   1:  PR[GP1:91,1] = PR[GP1:90,1] + -68.704;
   1:  PR[GP1:91,2] = PR[GP1:90,2] + 10.364;
   1:L PR[91] R[100]mm/sec CNT100;
   1:  PR[GP1:91,1] = PR[GP1:90,1] + -68.768;
   1:  PR[GP1:91,2] = PR[GP1:90,2] + 10.145;
   1:L PR[91] R[100]mm/sec CNT100;
   1:  PR[GP1:91,1] = PR[GP1:90,1] + -70.361;
   1:  PR[GP1:91,2] = PR[GP1:90,2] + -0.071;
   1:L PR[91] R[100]mm/sec CNT100;
   1:  PR[GP1:91,1] = PR[GP1:90,1] + -68.787;
   1:  PR[GP1:91,2] = PR[GP1:90,2] + -10.040;
   1:L PR[91] R[100]mm/sec CNT100;
   1:  PR[GP1:91,1] = PR[GP1:90,1] + -68.763;
   1:  PR[GP1:91,2] = PR[GP1:90,2] + -10.308;
   1:L PR[91] R[100]mm/sec CNT100;
   1:  PR[GP1:91,1] = PR[GP1:90,1] + -68.704;
   1:  PR[GP1:91,2] = PR[GP1:90,2] + -10.508;
   1:L PR[91] R[100]mm/sec CNT100;
   1:  PR[GP1:91,1] = PR[GP1:90,1] + -64.096;
   1:  PR[GP1:91,2] = PR[GP1:90,2] + -19.722;
   1:L PR[91] R[100]mm/sec CNT100;
   1:  PR[GP1:91,1] = PR[GP1:90,1] + -63.563;
   1:  PR[GP1:91,2] = PR[GP1:90,2] + -20.414;
   1:L PR[91] R[100]mm/sec CNT100;
   1:  PR[GP1:91,1] = PR[GP1:90,1] + -57.623;
   1:  PR[GP1:91,2] = PR[GP1:90,2] + -26.659;
   1:L PR[91] R[100]mm/sec CNT100;
   1:  PR[GP1:91,1] = PR[GP1:90,1] + -56.395;
   1:  PR[GP1:91,2] = PR[GP1:90,2] + -27.760;
   1:L PR[91] R[100]mm/sec CNT100;
   1:  PR[GP1:91,1] = PR[GP1:90,1] + -50.541;
   1:  PR[GP1:91,2] = PR[GP1:90,2] + -31.053;
   1:L PR[91] R[100]mm/sec CNT100;
   1:  PR[GP1:91,1] = PR[GP1:90,1] + -48.442;
   1:  PR[GP1:91,2] = PR[GP1:90,2] + -32.383;
   1:L PR[91] R[100]mm/sec CNT100;
   1:  PR[GP1:91,1] = PR[GP1:90,1] + -45.404;
   1:  PR[GP1:91,2] = PR[GP1:90,2] + -33.579;
   1:L PR[91] R[100]mm/sec CNT100;
   1:  PR[GP1:91,1] = PR[GP1:90,1] + -41.020;
   1:  PR[GP1:91,2] = PR[GP1:90,2] + -34.610;
   1:L PR[91] R[100]mm/sec CNT100;
   1:  PR[GP1:91,1] = PR[GP1:90,1] + -37.021;
   1:  PR[GP1:91,2] = PR[GP1:90,2] + -35.453;
   1:L PR[91] R[100]mm/sec CNT100;
   1:  PR[GP1:91,1] = PR[GP1:90,1] + -31.107;
   1:  PR[GP1:91,2] = PR[GP1:90,2] + -35.621;
   1:L PR[91] R[100]mm/sec CNT100;
   1:  PR[GP1:91,1] = PR[GP1:90,1] + -30.091;
   1:  PR[GP1:91,2] = PR[GP1:90,2] + -35.570;
   1:L PR[91] R[100]mm/sec CNT100;
   1:  PR[GP1:91,1] = PR[GP1:90,1] + -27.280;
   1:  PR[GP1:91,2] = PR[GP1:90,2] + -35.161;
   1:L PR[91] R[100]mm/sec CNT100;
   1:  PR[GP1:91,1] = PR[GP1:90,1] + -23.789;
   1:  PR[GP1:91,2] = PR[GP1:90,2] + -34.705;
   1:L PR[91] R[100]mm/sec CNT100;
   1:  PR[GP1:91,1] = PR[GP1:90,1] + -17.856;
   1:  PR[GP1:91,2] = PR[GP1:90,2] + -32.817;
   1:L PR[91] R[100]mm/sec CNT100;
   1:  PR[GP1:91,1] = PR[GP1:90,1] + -16.773;
   1:  PR[GP1:91,2] = PR[GP1:90,2] + -32.440;
   1:L PR[91] R[100]mm/sec CNT100;
   1:  PR[GP1:91,1] = PR[GP1:90,1] + -11.344;
   1:  PR[GP1:91,2] = PR[GP1:90,2] + -29.600;
   1:L PR[91] R[100]mm/sec CNT100;
   1:  PR[GP1:91,1] = PR[GP1:90,1] + -10.310;
   1:  PR[GP1:91,2] = PR[GP1:90,2] + -28.848;
   1:L PR[91] R[100]mm/sec CNT100;
   1:  PR[GP1:91,1] = PR[GP1:90,1] + -6.534;
   1:  PR[GP1:91,2] = PR[GP1:90,2] + -25.891;
   1:L PR[91] R[100]mm/sec CNT100;
   1:  PR[GP1:91,1] = PR[GP1:90,1] + -3.696;
   1:  PR[GP1:91,2] = PR[GP1:90,2] + -22.600;
   1:L PR[91] R[100]mm/sec CNT100;
   1:  PR[GP1:91,1] = PR[GP1:90,1] + -2.135;
   1:  PR[GP1:91,2] = PR[GP1:90,2] + -22.265;
   1:L PR[91] R[100]mm/sec CNT100;
   1:  PR[GP1:91,1] = PR[GP1:90,1] + 0.475;
   1:  PR[GP1:91,2] = PR[GP1:90,2] + -20.882;
   1:L PR[91] R[100]mm/sec CNT100;
   1:  PR[GP1:91,1] = PR[GP1:90,1] + 3.972;
   1:  PR[GP1:91,2] = PR[GP1:90,2] + -22.663;
   1:L PR[91] R[100]mm/sec CNT100;
   1:  PR[GP1:91,1] = PR[GP1:90,1] + 6.781;
   1:  PR[GP1:91,2] = PR[GP1:90,2] + -25.925;
   1:L PR[91] R[100]mm/sec CNT100;
   1:  PR[GP1:91,1] = PR[GP1:90,1] + 10.539;
   1:  PR[GP1:91,2] = PR[GP1:90,2] + -28.865;
   1:L PR[91] R[100]mm/sec CNT100;
   1:  PR[GP1:91,1] = PR[GP1:90,1] + 11.575;
   1:  PR[GP1:91,2] = PR[GP1:90,2] + -29.617;
   1:L PR[91] R[100]mm/sec CNT100;
   1:  PR[GP1:91,1] = PR[GP1:90,1] + 16.965;
   1:  PR[GP1:91,2] = PR[GP1:90,2] + -32.430;
   1:L PR[91] R[100]mm/sec CNT100;
   1:  PR[GP1:91,1] = PR[GP1:90,1] + 23.998;
   1:  PR[GP1:91,2] = PR[GP1:90,2] + -34.701;
   1:L PR[91] R[100]mm/sec CNT100;
   1:  PR[GP1:91,1] = PR[GP1:90,1] + 27.494;
   1:  PR[GP1:91,2] = PR[GP1:90,2] + -35.160;
   1:L PR[91] R[100]mm/sec CNT100;
   1:  PR[GP1:91,1] = PR[GP1:90,1] + 30.293;
   1:  PR[GP1:91,2] = PR[GP1:90,2] + -35.570;
   1:L PR[91] R[100]mm/sec CNT100;
   1:  PR[GP1:91,1] = PR[GP1:90,1] + 31.306;
   1:  PR[GP1:91,2] = PR[GP1:90,2] + -35.621;
   1:L PR[91] R[100]mm/sec CNT100;
   1:  PR[GP1:91,1] = PR[GP1:90,1] + 37.198;
   1:  PR[GP1:91,2] = PR[GP1:90,2] + -35.458;
   1:L PR[91] R[100]mm/sec CNT100;
   1:  PR[GP1:91,1] = PR[GP1:90,1] + 40.845;
   1:  PR[GP1:91,2] = PR[GP1:90,2] + -34.609;
   1:L PR[91] R[100]mm/sec CNT100;
   1:  PR[GP1:91,1] = PR[GP1:90,1] + 45.595;
   1:  PR[GP1:91,2] = PR[GP1:90,2] + -33.581;
   1:L PR[91] R[100]mm/sec CNT100;
   1:  PR[GP1:91,1] = PR[GP1:90,1] + 48.654;
   1:  PR[GP1:91,2] = PR[GP1:90,2] + -32.384;
   1:L PR[91] R[100]mm/sec CNT100;
   1:  PR[GP1:91,1] = PR[GP1:90,1] + 54.661;
   1:  PR[GP1:91,2] = PR[GP1:90,2] + -28.971;
   1:L PR[91] R[100]mm/sec CNT100;
   1:  PR[GP1:91,1] = PR[GP1:90,1] + 56.580;
   1:  PR[GP1:91,2] = PR[GP1:90,2] + -27.789;
   1:L PR[91] R[100]mm/sec CNT100;
   1:  PR[GP1:91,1] = PR[GP1:90,1] + 57.816;
   1:  PR[GP1:91,2] = PR[GP1:90,2] + -26.683;
   1:L PR[91] R[100]mm/sec CNT100;
   1:  PR[GP1:91,1] = PR[GP1:90,1] + 63.762;
   1:  PR[GP1:91,2] = PR[GP1:90,2] + -20.413;
   1:L PR[91] R[100]mm/sec CNT100;
   1:  PR[GP1:91,1] = PR[GP1:90,1] + 64.305;
   1:  PR[GP1:91,2] = PR[GP1:90,2] + -19.711;
   1:L PR[91] R[100]mm/sec CNT100;
   1:  PR[GP1:91,1] = PR[GP1:90,1] + 68.916;
   1:  PR[GP1:91,2] = PR[GP1:90,2] + -10.539;
   1:L PR[91] R[100]mm/sec CNT100;
   1:  PR[GP1:91,1] = PR[GP1:90,1] + 68.980;
   1:  PR[GP1:91,2] = PR[GP1:90,2] + -10.324;
   1:L PR[91] R[100]mm/sec CNT100;
   1:  PR[GP1:91,1] = PR[GP1:90,1] + 70.574;
   1:  PR[GP1:91,2] = PR[GP1:90,2] + -0.073;
   1:L PR[91] R[100]mm/sec CNT100;
   1:  PR[GP1:91,1] = PR[GP1:90,1] + 69.000;
   1:  PR[GP1:91,2] = PR[GP1:90,2] + 9.923;
   1:L PR[91] R[100]mm/sec CNT100;
   1:  PR[GP1:91,1] = PR[GP1:90,1] + 68.975;
   1:  PR[GP1:91,2] = PR[GP1:90,2] + 10.199;
   1:L PR[91] R[100]mm/sec CNT100;
   1:  PR[GP1:91,1] = PR[GP1:90,1] + 68.916;
   1:  PR[GP1:91,2] = PR[GP1:90,2] + 10.395;
   1:L PR[91] R[100]mm/sec CNT100;
   1:  PR[GP1:91,1] = PR[GP1:90,1] + 64.305;
   1:  PR[GP1:91,2] = PR[GP1:90,2] + 19.567;
   1:L PR[91] R[100]mm/sec CNT100;
   1:  PR[GP1:91,1] = PR[GP1:90,1] + 63.762;
   1:  PR[GP1:91,2] = PR[GP1:90,2] + 20.269;
   1:L PR[91] R[100]mm/sec CNT100;
   1:  PR[GP1:91,1] = PR[GP1:90,1] + 57.816;
   1:  PR[GP1:91,2] = PR[GP1:90,2] + 26.539;
   1:L PR[91] R[100]mm/sec CNT100;
   1:  PR[GP1:91,1] = PR[GP1:90,1] + 56.589;
   1:  PR[GP1:91,2] = PR[GP1:90,2] + 27.636;
   1:L PR[91] R[100]mm/sec CNT100;
   1:  PR[GP1:91,1] = PR[GP1:90,1] + 50.734;
   1:  PR[GP1:91,2] = PR[GP1:90,2] + 30.926;
   1:L PR[91] R[100]mm/sec CNT100;
   1:  PR[GP1:91,1] = PR[GP1:90,1] + 48.641;
   1:  PR[GP1:91,2] = PR[GP1:90,2] + 32.245;
   1:L PR[91] R[100]mm/sec CNT100;
   1:  PR[GP1:91,1] = PR[GP1:90,1] + 45.590;
   1:  PR[GP1:91,2] = PR[GP1:90,2] + 33.439;
   1:L PR[91] R[100]mm/sec CNT100;
   1:  PR[GP1:91,1] = PR[GP1:90,1] + 41.209;
   1:  PR[GP1:91,2] = PR[GP1:90,2] + 34.472;
   1:L PR[91] R[100]mm/sec CNT100;
   1:  PR[GP1:91,1] = PR[GP1:90,1] + 37.204;
   1:  PR[GP1:91,2] = PR[GP1:90,2] + 35.314;
   1:L PR[91] R[100]mm/sec CNT100;
   1:  PR[GP1:91,1] = PR[GP1:90,1] + 31.306;
   1:  PR[GP1:91,2] = PR[GP1:90,2] + 35.477;
   1:L PR[91] R[100]mm/sec CNT100;
   1:  PR[GP1:91,1] = PR[GP1:90,1] + 30.293;
   1:  PR[GP1:91,2] = PR[GP1:90,2] + 35.426;
   1:L PR[91] R[100]mm/sec CNT100;
   1:  PR[GP1:91,1] = PR[GP1:90,1] + 27.494;
   1:  PR[GP1:91,2] = PR[GP1:90,2] + 35.016;
   1:L PR[91] R[100]mm/sec CNT100;
   1:  PR[GP1:91,1] = PR[GP1:90,1] + 23.998;
   1:  PR[GP1:91,2] = PR[GP1:90,2] + 34.557;
   1:L PR[91] R[100]mm/sec CNT100;
   1:  PR[GP1:91,1] = PR[GP1:90,1] + 18.058;
   1:  PR[GP1:91,2] = PR[GP1:90,2] + 32.667;
   1:L PR[91] R[100]mm/sec CNT100;
   1:  PR[GP1:91,1] = PR[GP1:90,1] + 16.973;
   1:  PR[GP1:91,2] = PR[GP1:90,2] + 32.291;
   1:L PR[91] R[100]mm/sec CNT100;
   1:  PR[GP1:91,1] = PR[GP1:90,1] + 11.573;
   1:  PR[GP1:91,2] = PR[GP1:90,2] + 29.473;
   1:L PR[91] R[100]mm/sec CNT100;
   1:  PR[GP1:91,1] = PR[GP1:90,1] + 10.831;
   1:  PR[GP1:91,2] = PR[GP1:90,2] + 28.949;
   1:L PR[91] R[100]mm/sec CNT100;
   1:  PR[GP1:91,1] = PR[GP1:90,1] + 6.935;
   1:  PR[GP1:91,2] = PR[GP1:90,2] + 25.900;
   1:L PR[91] R[100]mm/sec CNT100;
   1:  PR[GP1:91,1] = PR[GP1:90,1] + 3.954;
   1:  PR[GP1:91,2] = PR[GP1:90,2] + 22.430;
   1:L PR[91] R[100]mm/sec CNT100;
   1:  PR[GP1:91,1] = PR[GP1:90,1] + 3.223;
   1:  PR[GP1:91,2] = PR[GP1:90,2] + 22.142;
   1:L PR[91] R[100]mm/sec CNT100;
   1:  PR[GP1:91,1] = PR[GP1:90,1] + 0.588;
   1:  PR[GP1:91,2] = PR[GP1:90,2] + 20.795;
   1:L PR[91] R[100]mm/sec CNT100;
   1:  ! -- Layer/Ebene 72 -- !;
   1:  PR[91] = PR[90];
   1:  PR[GP1:91,1] = PR[GP1:90,1] + -0.946;
   1:  PR[GP1:91,2] = PR[GP1:90,2] + 21.328;
   1:  PR[GP1:91,3] = PR[GP1:90,3] + 44.225;
   1:L PR[91] R[100]mm/sec CNT100;
   1:  PR[GP1:91,1] = PR[GP1:90,1] + -3.723;
   1:  PR[GP1:91,2] = PR[GP1:90,2] + 22.740;
   1:L PR[91] R[100]mm/sec CNT100;
   1:  PR[GP1:91,1] = PR[GP1:90,1] + -6.531;
   1:  PR[GP1:91,2] = PR[GP1:90,2] + 26.005;
   1:L PR[91] R[100]mm/sec CNT100;
   1:  PR[GP1:91,1] = PR[GP1:90,1] + -10.272;
   1:  PR[GP1:91,2] = PR[GP1:90,2] + 28.935;
   1:L PR[91] R[100]mm/sec CNT100;
   1:  PR[GP1:91,1] = PR[GP1:90,1] + -11.131;
   1:  PR[GP1:91,2] = PR[GP1:90,2] + 29.542;
   1:L PR[91] R[100]mm/sec CNT100;
   1:  PR[GP1:91,1] = PR[GP1:90,1] + -16.427;
   1:  PR[GP1:91,2] = PR[GP1:90,2] + 32.313;
   1:L PR[91] R[100]mm/sec CNT100;
   1:  PR[GP1:91,1] = PR[GP1:90,1] + -22.908;
   1:  PR[GP1:91,2] = PR[GP1:90,2] + 34.395;
   1:L PR[91] R[100]mm/sec CNT100;
   1:  PR[GP1:91,1] = PR[GP1:90,1] + -23.599;
   1:  PR[GP1:91,2] = PR[GP1:90,2] + 34.634;
   1:L PR[91] R[100]mm/sec CNT100;
   1:  PR[GP1:91,1] = PR[GP1:90,1] + -30.227;
   1:  PR[GP1:91,2] = PR[GP1:90,2] + 35.511;
   1:L PR[91] R[100]mm/sec CNT100;
   1:  PR[GP1:91,1] = PR[GP1:90,1] + -30.457;
   1:  PR[GP1:91,2] = PR[GP1:90,2] + 35.523;
   1:L PR[91] R[100]mm/sec CNT100;
   1:  PR[GP1:91,1] = PR[GP1:90,1] + -36.896;
   1:  PR[GP1:91,2] = PR[GP1:90,2] + 35.340;
   1:L PR[91] R[100]mm/sec CNT100;
   1:  PR[GP1:91,1] = PR[GP1:90,1] + -39.667;
   1:  PR[GP1:91,2] = PR[GP1:90,2] + 34.695;
   1:L PR[91] R[100]mm/sec CNT100;
   1:  PR[GP1:91,1] = PR[GP1:90,1] + -45.015;
   1:  PR[GP1:91,2] = PR[GP1:90,2] + 33.536;
   1:L PR[91] R[100]mm/sec CNT100;
   1:  PR[GP1:91,1] = PR[GP1:90,1] + -48.459;
   1:  PR[GP1:91,2] = PR[GP1:90,2] + 32.181;
   1:L PR[91] R[100]mm/sec CNT100;
   1:  PR[GP1:91,1] = PR[GP1:90,1] + -53.838;
   1:  PR[GP1:91,2] = PR[GP1:90,2] + 29.120;
   1:L PR[91] R[100]mm/sec CNT100;
   1:  PR[GP1:91,1] = PR[GP1:90,1] + -56.172;
   1:  PR[GP1:91,2] = PR[GP1:90,2] + 27.675;
   1:L PR[91] R[100]mm/sec CNT100;
   1:  PR[GP1:91,1] = PR[GP1:90,1] + -57.679;
   1:  PR[GP1:91,2] = PR[GP1:90,2] + 26.324;
   1:L PR[91] R[100]mm/sec CNT100;
   1:  PR[GP1:91,1] = PR[GP1:90,1] + -63.196;
   1:  PR[GP1:91,2] = PR[GP1:90,2] + 20.524;
   1:L PR[91] R[100]mm/sec CNT100;
   1:  PR[GP1:91,1] = PR[GP1:90,1] + -63.972;
   1:  PR[GP1:91,2] = PR[GP1:90,2] + 19.517;
   1:L PR[91] R[100]mm/sec CNT100;
   1:  PR[GP1:91,1] = PR[GP1:90,1] + -68.487;
   1:  PR[GP1:91,2] = PR[GP1:90,2] + 10.491;
   1:L PR[91] R[100]mm/sec CNT100;
   1:  PR[GP1:91,1] = PR[GP1:90,1] + -68.652;
   1:  PR[GP1:91,2] = PR[GP1:90,2] + 9.931;
   1:L PR[91] R[100]mm/sec CNT100;
   1:  PR[GP1:91,1] = PR[GP1:90,1] + -70.166;
   1:  PR[GP1:91,2] = PR[GP1:90,2] + 0.222;
   1:L PR[91] R[100]mm/sec CNT100;
   1:  PR[GP1:91,1] = PR[GP1:90,1] + -70.190;
   1:  PR[GP1:91,2] = PR[GP1:90,2] + -0.052;
   1:L PR[91] R[100]mm/sec CNT100;
   1:  PR[GP1:91,1] = PR[GP1:90,1] + -68.700;
   1:  PR[GP1:91,2] = PR[GP1:90,2] + -9.487;
   1:L PR[91] R[100]mm/sec CNT100;
   1:  PR[GP1:91,1] = PR[GP1:90,1] + -68.646;
   1:  PR[GP1:91,2] = PR[GP1:90,2] + -10.094;
   1:L PR[91] R[100]mm/sec CNT100;
   1:  PR[GP1:91,1] = PR[GP1:90,1] + -68.487;
   1:  PR[GP1:91,2] = PR[GP1:90,2] + -10.635;
   1:L PR[91] R[100]mm/sec CNT100;
   1:  PR[GP1:91,1] = PR[GP1:90,1] + -63.972;
   1:  PR[GP1:91,2] = PR[GP1:90,2] + -19.661;
   1:L PR[91] R[100]mm/sec CNT100;
   1:  PR[GP1:91,1] = PR[GP1:90,1] + -63.196;
   1:  PR[GP1:91,2] = PR[GP1:90,2] + -20.668;
   1:L PR[91] R[100]mm/sec CNT100;
   1:  PR[GP1:91,1] = PR[GP1:90,1] + -57.679;
   1:  PR[GP1:91,2] = PR[GP1:90,2] + -26.468;
   1:L PR[91] R[100]mm/sec CNT100;
   1:  PR[GP1:91,1] = PR[GP1:90,1] + -56.181;
   1:  PR[GP1:91,2] = PR[GP1:90,2] + -27.810;
   1:L PR[91] R[100]mm/sec CNT100;
   1:  PR[GP1:91,1] = PR[GP1:90,1] + -50.817;
   1:  PR[GP1:91,2] = PR[GP1:90,2] + -30.828;
   1:L PR[91] R[100]mm/sec CNT100;
   1:  PR[GP1:91,1] = PR[GP1:90,1] + -48.446;
   1:  PR[GP1:91,2] = PR[GP1:90,2] + -32.330;
   1:L PR[91] R[100]mm/sec CNT100;
   1:  PR[GP1:91,1] = PR[GP1:90,1] + -45.010;
   1:  PR[GP1:91,2] = PR[GP1:90,2] + -33.682;
   1:L PR[91] R[100]mm/sec CNT100;
   1:  PR[GP1:91,1] = PR[GP1:90,1] + -41.261;
   1:  PR[GP1:91,2] = PR[GP1:90,2] + -34.565;
   1:L PR[91] R[100]mm/sec CNT100;
   1:  PR[GP1:91,1] = PR[GP1:90,1] + -36.902;
   1:  PR[GP1:91,2] = PR[GP1:90,2] + -35.483;
   1:L PR[91] R[100]mm/sec CNT100;
   1:  PR[GP1:91,1] = PR[GP1:90,1] + -30.457;
   1:  PR[GP1:91,2] = PR[GP1:90,2] + -35.667;
   1:L PR[91] R[100]mm/sec CNT100;
   1:  PR[GP1:91,1] = PR[GP1:90,1] + -30.227;
   1:  PR[GP1:91,2] = PR[GP1:90,2] + -35.655;
   1:L PR[91] R[100]mm/sec CNT100;
   1:  PR[GP1:91,1] = PR[GP1:90,1] + -23.591;
   1:  PR[GP1:91,2] = PR[GP1:90,2] + -34.777;
   1:L PR[91] R[100]mm/sec CNT100;
   1:  PR[GP1:91,1] = PR[GP1:90,1] + -17.788;
   1:  PR[GP1:91,2] = PR[GP1:90,2] + -32.930;
   1:L PR[91] R[100]mm/sec CNT100;
   1:  PR[GP1:91,1] = PR[GP1:90,1] + -16.431;
   1:  PR[GP1:91,2] = PR[GP1:90,2] + -32.459;
   1:L PR[91] R[100]mm/sec CNT100;
   1:  PR[GP1:91,1] = PR[GP1:90,1] + -11.133;
   1:  PR[GP1:91,2] = PR[GP1:90,2] + -29.687;
   1:L PR[91] R[100]mm/sec CNT100;
   1:  PR[GP1:91,1] = PR[GP1:90,1] + -9.935;
   1:  PR[GP1:91,2] = PR[GP1:90,2] + -28.817;
   1:L PR[91] R[100]mm/sec CNT100;
   1:  PR[GP1:91,1] = PR[GP1:90,1] + -6.361;
   1:  PR[GP1:91,2] = PR[GP1:90,2] + -26.017;
   1:L PR[91] R[100]mm/sec CNT100;
   1:  PR[GP1:91,1] = PR[GP1:90,1] + -3.667;
   1:  PR[GP1:91,2] = PR[GP1:90,2] + -22.893;
   1:L PR[91] R[100]mm/sec CNT100;
   1:  PR[GP1:91,1] = PR[GP1:90,1] + -1.968;
   1:  PR[GP1:91,2] = PR[GP1:90,2] + -22.529;
   1:L PR[91] R[100]mm/sec CNT100;
   1:  PR[GP1:91,1] = PR[GP1:90,1] + 0.517;
   1:  PR[GP1:91,2] = PR[GP1:90,2] + -21.212;
   1:L PR[91] R[100]mm/sec CNT100;
   1:  PR[GP1:91,1] = PR[GP1:90,1] + 3.942;
   1:  PR[GP1:91,2] = PR[GP1:90,2] + -22.956;
   1:L PR[91] R[100]mm/sec CNT100;
   1:  PR[GP1:91,1] = PR[GP1:90,1] + 6.606;
   1:  PR[GP1:91,2] = PR[GP1:90,2] + -26.049;
   1:L PR[91] R[100]mm/sec CNT100;
   1:  PR[GP1:91,1] = PR[GP1:90,1] + 10.164;
   1:  PR[GP1:91,2] = PR[GP1:90,2] + -28.833;
   1:L PR[91] R[100]mm/sec CNT100;
   1:  PR[GP1:91,1] = PR[GP1:90,1] + 11.363;
   1:  PR[GP1:91,2] = PR[GP1:90,2] + -29.704;
   1:L PR[91] R[100]mm/sec CNT100;
   1:  PR[GP1:91,1] = PR[GP1:90,1] + 16.623;
   1:  PR[GP1:91,2] = PR[GP1:90,2] + -32.449;
   1:L PR[91] R[100]mm/sec CNT100;
   1:  PR[GP1:91,1] = PR[GP1:90,1] + 23.114;
   1:  PR[GP1:91,2] = PR[GP1:90,2] + -34.534;
   1:L PR[91] R[100]mm/sec CNT100;
   1:  PR[GP1:91,1] = PR[GP1:90,1] + 23.806;
   1:  PR[GP1:91,2] = PR[GP1:90,2] + -34.774;
   1:L PR[91] R[100]mm/sec CNT100;
   1:  PR[GP1:91,1] = PR[GP1:90,1] + 30.428;
   1:  PR[GP1:91,2] = PR[GP1:90,2] + -35.655;
   1:L PR[91] R[100]mm/sec CNT100;
   1:  PR[GP1:91,1] = PR[GP1:90,1] + 30.654;
   1:  PR[GP1:91,2] = PR[GP1:90,2] + -35.667;
   1:L PR[91] R[100]mm/sec CNT100;
   1:  PR[GP1:91,1] = PR[GP1:90,1] + 37.075;
   1:  PR[GP1:91,2] = PR[GP1:90,2] + -35.488;
   1:L PR[91] R[100]mm/sec CNT100;
   1:  PR[GP1:91,1] = PR[GP1:90,1] + 39.837;
   1:  PR[GP1:91,2] = PR[GP1:90,2] + -34.846;
   1:L PR[91] R[100]mm/sec CNT100;
   1:  PR[GP1:91,1] = PR[GP1:90,1] + 45.197;
   1:  PR[GP1:91,2] = PR[GP1:90,2] + -33.686;
   1:L PR[91] R[100]mm/sec CNT100;
   1:  PR[GP1:91,1] = PR[GP1:90,1] + 48.657;
   1:  PR[GP1:91,2] = PR[GP1:90,2] + -32.332;
   1:L PR[91] R[100]mm/sec CNT100;
   1:  PR[GP1:91,1] = PR[GP1:90,1] + 54.035;
   1:  PR[GP1:91,2] = PR[GP1:90,2] + -29.277;
   1:L PR[91] R[100]mm/sec CNT100;
   1:  PR[GP1:91,1] = PR[GP1:90,1] + 56.363;
   1:  PR[GP1:91,2] = PR[GP1:90,2] + -27.841;
   1:L PR[91] R[100]mm/sec CNT100;
   1:  PR[GP1:91,1] = PR[GP1:90,1] + 57.868;
   1:  PR[GP1:91,2] = PR[GP1:90,2] + -26.496;
   1:L PR[91] R[100]mm/sec CNT100;
   1:  PR[GP1:91,1] = PR[GP1:90,1] + 63.389;
   1:  PR[GP1:91,2] = PR[GP1:90,2] + -20.673;
   1:L PR[91] R[100]mm/sec CNT100;
   1:  PR[GP1:91,1] = PR[GP1:90,1] + 64.178;
   1:  PR[GP1:91,2] = PR[GP1:90,2] + -19.653;
   1:L PR[91] R[100]mm/sec CNT100;
   1:  PR[GP1:91,1] = PR[GP1:90,1] + 68.698;
   1:  PR[GP1:91,2] = PR[GP1:90,2] + -10.669;
   1:L PR[91] R[100]mm/sec CNT100;
   1:  PR[GP1:91,1] = PR[GP1:90,1] + 68.862;
   1:  PR[GP1:91,2] = PR[GP1:90,2] + -10.118;
   1:L PR[91] R[100]mm/sec CNT100;
   1:  PR[GP1:91,1] = PR[GP1:90,1] + 70.377;
   1:  PR[GP1:91,2] = PR[GP1:90,2] + -0.376;
   1:L PR[91] R[100]mm/sec CNT100;
   1:  PR[GP1:91,1] = PR[GP1:90,1] + 70.403;
   1:  PR[GP1:91,2] = PR[GP1:90,2] + -0.092;
   1:L PR[91] R[100]mm/sec CNT100;
   1:  PR[GP1:91,1] = PR[GP1:90,1] + 68.913;
   1:  PR[GP1:91,2] = PR[GP1:90,2] + 9.368;
   1:L PR[91] R[100]mm/sec CNT100;
   1:  PR[GP1:91,1] = PR[GP1:90,1] + 68.857;
   1:  PR[GP1:91,2] = PR[GP1:90,2] + 9.993;
   1:L PR[91] R[100]mm/sec CNT100;
   1:  PR[GP1:91,1] = PR[GP1:90,1] + 68.698;
   1:  PR[GP1:91,2] = PR[GP1:90,2] + 10.525;
   1:L PR[91] R[100]mm/sec CNT100;
   1:  PR[GP1:91,1] = PR[GP1:90,1] + 64.178;
   1:  PR[GP1:91,2] = PR[GP1:90,2] + 19.509;
   1:L PR[91] R[100]mm/sec CNT100;
   1:  PR[GP1:91,1] = PR[GP1:90,1] + 63.389;
   1:  PR[GP1:91,2] = PR[GP1:90,2] + 20.529;
   1:L PR[91] R[100]mm/sec CNT100;
   1:  PR[GP1:91,1] = PR[GP1:90,1] + 57.868;
   1:  PR[GP1:91,2] = PR[GP1:90,2] + 26.352;
   1:L PR[91] R[100]mm/sec CNT100;
   1:  PR[GP1:91,1] = PR[GP1:90,1] + 56.372;
   1:  PR[GP1:91,2] = PR[GP1:90,2] + 27.689;
   1:L PR[91] R[100]mm/sec CNT100;
   1:  PR[GP1:91,1] = PR[GP1:90,1] + 51.007;
   1:  PR[GP1:91,2] = PR[GP1:90,2] + 30.704;
   1:L PR[91] R[100]mm/sec CNT100;
   1:  PR[GP1:91,1] = PR[GP1:90,1] + 48.644;
   1:  PR[GP1:91,2] = PR[GP1:90,2] + 32.193;
   1:L PR[91] R[100]mm/sec CNT100;
   1:  PR[GP1:91,1] = PR[GP1:90,1] + 45.192;
   1:  PR[GP1:91,2] = PR[GP1:90,2] + 33.544;
   1:L PR[91] R[100]mm/sec CNT100;
   1:  PR[GP1:91,1] = PR[GP1:90,1] + 41.447;
   1:  PR[GP1:91,2] = PR[GP1:90,2] + 34.427;
   1:L PR[91] R[100]mm/sec CNT100;
   1:  PR[GP1:91,1] = PR[GP1:90,1] + 37.082;
   1:  PR[GP1:91,2] = PR[GP1:90,2] + 35.344;
   1:L PR[91] R[100]mm/sec CNT100;
   1:  PR[GP1:91,1] = PR[GP1:90,1] + 30.654;
   1:  PR[GP1:91,2] = PR[GP1:90,2] + 35.523;
   1:L PR[91] R[100]mm/sec CNT100;
   1:  PR[GP1:91,1] = PR[GP1:90,1] + 30.428;
   1:  PR[GP1:91,2] = PR[GP1:90,2] + 35.511;
   1:L PR[91] R[100]mm/sec CNT100;
   1:  PR[GP1:91,1] = PR[GP1:90,1] + 23.800;
   1:  PR[GP1:91,2] = PR[GP1:90,2] + 34.629;
   1:L PR[91] R[100]mm/sec CNT100;
   1:  PR[GP1:91,1] = PR[GP1:90,1] + 17.990;
   1:  PR[GP1:91,2] = PR[GP1:90,2] + 32.781;
   1:L PR[91] R[100]mm/sec CNT100;
   1:  PR[GP1:91,1] = PR[GP1:90,1] + 16.631;
   1:  PR[GP1:91,2] = PR[GP1:90,2] + 32.309;
   1:L PR[91] R[100]mm/sec CNT100;
   1:  PR[GP1:91,1] = PR[GP1:90,1] + 11.361;
   1:  PR[GP1:91,2] = PR[GP1:90,2] + 29.559;
   1:L PR[91] R[100]mm/sec CNT100;
   1:  PR[GP1:91,1] = PR[GP1:90,1] + 10.500;
   1:  PR[GP1:91,2] = PR[GP1:90,2] + 28.951;
   1:L PR[91] R[100]mm/sec CNT100;
   1:  PR[GP1:91,1] = PR[GP1:90,1] + 6.777;
   1:  PR[GP1:91,2] = PR[GP1:90,2] + 26.038;
   1:L PR[91] R[100]mm/sec CNT100;
   1:  PR[GP1:91,1] = PR[GP1:90,1] + 3.924;
   1:  PR[GP1:91,2] = PR[GP1:90,2] + 22.717;
   1:L PR[91] R[100]mm/sec CNT100;
   1:  PR[GP1:91,1] = PR[GP1:90,1] + 3.134;
   1:  PR[GP1:91,2] = PR[GP1:90,2] + 22.405;
   1:L PR[91] R[100]mm/sec CNT100;
   1:  PR[GP1:91,1] = PR[GP1:90,1] + 0.630;
   1:  PR[GP1:91,2] = PR[GP1:90,2] + 21.125;
   1:L PR[91] R[100]mm/sec CNT100;
   1:  ! -- Layer/Ebene 73 -- !;
   1:  PR[91] = PR[90];
   1:  PR[GP1:91,1] = PR[GP1:90,1] + -1.034;
   1:  PR[GP1:91,2] = PR[GP1:90,2] + 21.674;
   1:  PR[GP1:91,3] = PR[GP1:90,3] + 44.835;
   1:L PR[91] R[100]mm/sec CNT100;
   1:  PR[GP1:91,1] = PR[GP1:90,1] + -3.694;
   1:  PR[GP1:91,2] = PR[GP1:90,2] + 23.027;
   1:L PR[91] R[100]mm/sec CNT100;
   1:  PR[GP1:91,1] = PR[GP1:90,1] + -6.375;
   1:  PR[GP1:91,2] = PR[GP1:90,2] + 26.144;
   1:L PR[91] R[100]mm/sec CNT100;
   1:  PR[GP1:91,1] = PR[GP1:90,1] + -9.942;
   1:  PR[GP1:91,2] = PR[GP1:90,2] + 28.938;
   1:L PR[91] R[100]mm/sec CNT100;
   1:  PR[GP1:91,1] = PR[GP1:90,1] + -10.921;
   1:  PR[GP1:91,2] = PR[GP1:90,2] + 29.630;
   1:L PR[91] R[100]mm/sec CNT100;
   1:  PR[GP1:91,1] = PR[GP1:90,1] + -16.085;
   1:  PR[GP1:91,2] = PR[GP1:90,2] + 32.332;
   1:L PR[91] R[100]mm/sec CNT100;
   1:  PR[GP1:91,1] = PR[GP1:90,1] + -22.408;
   1:  PR[GP1:91,2] = PR[GP1:90,2] + 34.363;
   1:L PR[91] R[100]mm/sec CNT100;
   1:  PR[GP1:91,1] = PR[GP1:90,1] + -23.400;
   1:  PR[GP1:91,2] = PR[GP1:90,2] + 34.706;
   1:L PR[91] R[100]mm/sec CNT100;
   1:  PR[GP1:91,1] = PR[GP1:90,1] + -30.023;
   1:  PR[GP1:91,2] = PR[GP1:90,2] + 35.572;
   1:L PR[91] R[100]mm/sec CNT100;
   1:  PR[GP1:91,1] = PR[GP1:90,1] + -36.775;
   1:  PR[GP1:91,2] = PR[GP1:90,2] + 35.370;
   1:L PR[91] R[100]mm/sec CNT100;
   1:  PR[GP1:91,1] = PR[GP1:90,1] + -38.664;
   1:  PR[GP1:91,2] = PR[GP1:90,2] + 34.931;
   1:L PR[91] R[100]mm/sec CNT100;
   1:  PR[GP1:91,1] = PR[GP1:90,1] + -44.621;
   1:  PR[GP1:91,2] = PR[GP1:90,2] + 33.640;
   1:L PR[91] R[100]mm/sec CNT100;
   1:  PR[GP1:91,1] = PR[GP1:90,1] + -48.464;
   1:  PR[GP1:91,2] = PR[GP1:90,2] + 32.128;
   1:L PR[91] R[100]mm/sec CNT100;
   1:  PR[GP1:91,1] = PR[GP1:90,1] + -53.214;
   1:  PR[GP1:91,2] = PR[GP1:90,2] + 29.425;
   1:L PR[91] R[100]mm/sec CNT100;
   1:  PR[GP1:91,1] = PR[GP1:90,1] + -55.959;
   1:  PR[GP1:91,2] = PR[GP1:90,2] + 27.724;
   1:L PR[91] R[100]mm/sec CNT100;
   1:  PR[GP1:91,1] = PR[GP1:90,1] + -57.735;
   1:  PR[GP1:91,2] = PR[GP1:90,2] + 26.132;
   1:L PR[91] R[100]mm/sec CNT100;
   1:  PR[GP1:91,1] = PR[GP1:90,1] + -62.829;
   1:  PR[GP1:91,2] = PR[GP1:90,2] + 20.777;
   1:L PR[91] R[100]mm/sec CNT100;
   1:  PR[GP1:91,1] = PR[GP1:90,1] + -63.847;
   1:  PR[GP1:91,2] = PR[GP1:90,2] + 19.455;
   1:L PR[91] R[100]mm/sec CNT100;
   1:  PR[GP1:91,1] = PR[GP1:90,1] + -68.270;
   1:  PR[GP1:91,2] = PR[GP1:90,2] + 10.617;
   1:L PR[91] R[100]mm/sec CNT100;
   1:  PR[GP1:91,1] = PR[GP1:90,1] + -68.535;
   1:  PR[GP1:91,2] = PR[GP1:90,2] + 9.717;
   1:L PR[91] R[100]mm/sec CNT100;
   1:  PR[GP1:91,1] = PR[GP1:90,1] + -69.959;
   1:  PR[GP1:91,2] = PR[GP1:90,2] + 0.585;
   1:L PR[91] R[100]mm/sec CNT100;
   1:  PR[GP1:91,1] = PR[GP1:90,1] + -70.016;
   1:  PR[GP1:91,2] = PR[GP1:90,2] + -0.052;
   1:L PR[91] R[100]mm/sec CNT100;
   1:  PR[GP1:91,1] = PR[GP1:90,1] + -68.613;
   1:  PR[GP1:91,2] = PR[GP1:90,2] + -8.933;
   1:L PR[91] R[100]mm/sec CNT100;
   1:  PR[GP1:91,1] = PR[GP1:90,1] + -68.530;
   1:  PR[GP1:91,2] = PR[GP1:90,2] + -9.880;
   1:L PR[91] R[100]mm/sec CNT100;
   1:  PR[GP1:91,1] = PR[GP1:90,1] + -68.270;
   1:  PR[GP1:91,2] = PR[GP1:90,2] + -10.761;
   1:L PR[91] R[100]mm/sec CNT100;
   1:  PR[GP1:91,1] = PR[GP1:90,1] + -63.847;
   1:  PR[GP1:91,2] = PR[GP1:90,2] + -19.599;
   1:L PR[91] R[100]mm/sec CNT100;
   1:  PR[GP1:91,1] = PR[GP1:90,1] + -62.829;
   1:  PR[GP1:91,2] = PR[GP1:90,2] + -20.921;
   1:L PR[91] R[100]mm/sec CNT100;
   1:  PR[GP1:91,1] = PR[GP1:90,1] + -57.735;
   1:  PR[GP1:91,2] = PR[GP1:90,2] + -26.276;
   1:L PR[91] R[100]mm/sec CNT100;
   1:  PR[GP1:91,1] = PR[GP1:90,1] + -55.968;
   1:  PR[GP1:91,2] = PR[GP1:90,2] + -27.860;
   1:L PR[91] R[100]mm/sec CNT100;
   1:  PR[GP1:91,1] = PR[GP1:90,1] + -51.092;
   1:  PR[GP1:91,2] = PR[GP1:90,2] + -30.603;
   1:L PR[91] R[100]mm/sec CNT100;
   1:  PR[GP1:91,1] = PR[GP1:90,1] + -48.450;
   1:  PR[GP1:91,2] = PR[GP1:90,2] + -32.277;
   1:L PR[91] R[100]mm/sec CNT100;
   1:  PR[GP1:91,1] = PR[GP1:90,1] + -44.616;
   1:  PR[GP1:91,2] = PR[GP1:90,2] + -33.786;
   1:L PR[91] R[100]mm/sec CNT100;
   1:  PR[GP1:91,1] = PR[GP1:90,1] + -41.501;
   1:  PR[GP1:91,2] = PR[GP1:90,2] + -34.519;
   1:L PR[91] R[100]mm/sec CNT100;
   1:  PR[GP1:91,1] = PR[GP1:90,1] + -36.782;
   1:  PR[GP1:91,2] = PR[GP1:90,2] + -35.514;
   1:L PR[91] R[100]mm/sec CNT100;
   1:  PR[GP1:91,1] = PR[GP1:90,1] + -30.023;
   1:  PR[GP1:91,2] = PR[GP1:90,2] + -35.716;
   1:L PR[91] R[100]mm/sec CNT100;
   1:  PR[GP1:91,1] = PR[GP1:90,1] + -23.391;
   1:  PR[GP1:91,2] = PR[GP1:90,2] + -34.849;
   1:L PR[91] R[100]mm/sec CNT100;
   1:  PR[GP1:91,1] = PR[GP1:90,1] + -17.719;
   1:  PR[GP1:91,2] = PR[GP1:90,2] + -33.044;
   1:L PR[91] R[100]mm/sec CNT100;
   1:  PR[GP1:91,1] = PR[GP1:90,1] + -16.089;
   1:  PR[GP1:91,2] = PR[GP1:90,2] + -32.477;
   1:L PR[91] R[100]mm/sec CNT100;
   1:  PR[GP1:91,1] = PR[GP1:90,1] + -10.922;
   1:  PR[GP1:91,2] = PR[GP1:90,2] + -29.774;
   1:L PR[91] R[100]mm/sec CNT100;
   1:  PR[GP1:91,1] = PR[GP1:90,1] + -9.561;
   1:  PR[GP1:91,2] = PR[GP1:90,2] + -28.785;
   1:L PR[91] R[100]mm/sec CNT100;
   1:  PR[GP1:91,1] = PR[GP1:90,1] + -6.187;
   1:  PR[GP1:91,2] = PR[GP1:90,2] + -26.143;
   1:L PR[91] R[100]mm/sec CNT100;
   1:  PR[GP1:91,1] = PR[GP1:90,1] + -3.638;
   1:  PR[GP1:91,2] = PR[GP1:90,2] + -23.186;
   1:L PR[91] R[100]mm/sec CNT100;
   1:  PR[GP1:91,1] = PR[GP1:90,1] + -1.801;
   1:  PR[GP1:91,2] = PR[GP1:90,2] + -22.792;
   1:L PR[91] R[100]mm/sec CNT100;
   1:  PR[GP1:91,1] = PR[GP1:90,1] + 0.558;
   1:  PR[GP1:91,2] = PR[GP1:90,2] + -21.542;
   1:L PR[91] R[100]mm/sec CNT100;
   1:  PR[GP1:91,1] = PR[GP1:90,1] + 3.912;
   1:  PR[GP1:91,2] = PR[GP1:90,2] + -23.249;
   1:L PR[91] R[100]mm/sec CNT100;
   1:  PR[GP1:91,1] = PR[GP1:90,1] + 6.430;
   1:  PR[GP1:91,2] = PR[GP1:90,2] + -26.173;
   1:L PR[91] R[100]mm/sec CNT100;
   1:  PR[GP1:91,1] = PR[GP1:90,1] + 9.788;
   1:  PR[GP1:91,2] = PR[GP1:90,2] + -28.801;
   1:L PR[91] R[100]mm/sec CNT100;
   1:  PR[GP1:91,1] = PR[GP1:90,1] + 11.151;
   1:  PR[GP1:91,2] = PR[GP1:90,2] + -29.791;
   1:L PR[91] R[100]mm/sec CNT100;
   1:  PR[GP1:91,1] = PR[GP1:90,1] + 16.280;
   1:  PR[GP1:91,2] = PR[GP1:90,2] + -32.468;
   1:L PR[91] R[100]mm/sec CNT100;
   1:  PR[GP1:91,1] = PR[GP1:90,1] + 22.612;
   1:  PR[GP1:91,2] = PR[GP1:90,2] + -34.502;
   1:L PR[91] R[100]mm/sec CNT100;
   1:  PR[GP1:91,1] = PR[GP1:90,1] + 23.607;
   1:  PR[GP1:91,2] = PR[GP1:90,2] + -34.846;
   1:L PR[91] R[100]mm/sec CNT100;
   1:  PR[GP1:91,1] = PR[GP1:90,1] + 30.222;
   1:  PR[GP1:91,2] = PR[GP1:90,2] + -35.716;
   1:L PR[91] R[100]mm/sec CNT100;
   1:  PR[GP1:91,1] = PR[GP1:90,1] + 36.952;
   1:  PR[GP1:91,2] = PR[GP1:90,2] + -35.519;
   1:L PR[91] R[100]mm/sec CNT100;
   1:  PR[GP1:91,1] = PR[GP1:90,1] + 38.829;
   1:  PR[GP1:91,2] = PR[GP1:90,2] + -35.082;
   1:L PR[91] R[100]mm/sec CNT100;
   1:  PR[GP1:91,1] = PR[GP1:90,1] + 44.799;
   1:  PR[GP1:91,2] = PR[GP1:90,2] + -33.791;
   1:L PR[91] R[100]mm/sec CNT100;
   1:  PR[GP1:91,1] = PR[GP1:90,1] + 48.659;
   1:  PR[GP1:91,2] = PR[GP1:90,2] + -32.280;
   1:L PR[91] R[100]mm/sec CNT100;
   1:  PR[GP1:91,1] = PR[GP1:90,1] + 53.408;
   1:  PR[GP1:91,2] = PR[GP1:90,2] + -29.582;
   1:L PR[91] R[100]mm/sec CNT100;
   1:  PR[GP1:91,1] = PR[GP1:90,1] + 56.146;
   1:  PR[GP1:91,2] = PR[GP1:90,2] + -27.894;
   1:L PR[91] R[100]mm/sec CNT100;
   1:  PR[GP1:91,1] = PR[GP1:90,1] + 57.920;
   1:  PR[GP1:91,2] = PR[GP1:90,2] + -26.309;
   1:L PR[91] R[100]mm/sec CNT100;
   1:  PR[GP1:91,1] = PR[GP1:90,1] + 63.017;
   1:  PR[GP1:91,2] = PR[GP1:90,2] + -20.933;
   1:L PR[91] R[100]mm/sec CNT100;
   1:  PR[GP1:91,1] = PR[GP1:90,1] + 64.051;
   1:  PR[GP1:91,2] = PR[GP1:90,2] + -19.595;
   1:L PR[91] R[100]mm/sec CNT100;
   1:  PR[GP1:91,1] = PR[GP1:90,1] + 68.479;
   1:  PR[GP1:91,2] = PR[GP1:90,2] + -10.799;
   1:L PR[91] R[100]mm/sec CNT100;
   1:  PR[GP1:91,1] = PR[GP1:90,1] + 68.744;
   1:  PR[GP1:91,2] = PR[GP1:90,2] + -9.912;
   1:L PR[91] R[100]mm/sec CNT100;
   1:  PR[GP1:91,1] = PR[GP1:90,1] + 70.169;
   1:  PR[GP1:91,2] = PR[GP1:90,2] + -0.749;
   1:L PR[91] R[100]mm/sec CNT100;
   1:  PR[GP1:91,1] = PR[GP1:90,1] + 70.229;
   1:  PR[GP1:91,2] = PR[GP1:90,2] + -0.092;
   1:L PR[91] R[100]mm/sec CNT100;
   1:  PR[GP1:91,1] = PR[GP1:90,1] + 68.827;
   1:  PR[GP1:91,2] = PR[GP1:90,2] + 8.814;
   1:L PR[91] R[100]mm/sec CNT100;
   1:  PR[GP1:91,1] = PR[GP1:90,1] + 68.739;
   1:  PR[GP1:91,2] = PR[GP1:90,2] + 9.786;
   1:L PR[91] R[100]mm/sec CNT100;
   1:  PR[GP1:91,1] = PR[GP1:90,1] + 68.479;
   1:  PR[GP1:91,2] = PR[GP1:90,2] + 10.655;
   1:L PR[91] R[100]mm/sec CNT100;
   1:  PR[GP1:91,1] = PR[GP1:90,1] + 64.051;
   1:  PR[GP1:91,2] = PR[GP1:90,2] + 19.451;
   1:L PR[91] R[100]mm/sec CNT100;
   1:  PR[GP1:91,1] = PR[GP1:90,1] + 63.017;
   1:  PR[GP1:91,2] = PR[GP1:90,2] + 20.789;
   1:L PR[91] R[100]mm/sec CNT100;
   1:  PR[GP1:91,1] = PR[GP1:90,1] + 57.920;
   1:  PR[GP1:91,2] = PR[GP1:90,2] + 26.165;
   1:L PR[91] R[100]mm/sec CNT100;
   1:  PR[GP1:91,1] = PR[GP1:90,1] + 56.155;
   1:  PR[GP1:91,2] = PR[GP1:90,2] + 27.742;
   1:L PR[91] R[100]mm/sec CNT100;
   1:  PR[GP1:91,1] = PR[GP1:90,1] + 51.280;
   1:  PR[GP1:91,2] = PR[GP1:90,2] + 30.481;
   1:L PR[91] R[100]mm/sec CNT100;
   1:  PR[GP1:91,1] = PR[GP1:90,1] + 48.646;
   1:  PR[GP1:91,2] = PR[GP1:90,2] + 32.141;
   1:L PR[91] R[100]mm/sec CNT100;
   1:  PR[GP1:91,1] = PR[GP1:90,1] + 44.794;
   1:  PR[GP1:91,2] = PR[GP1:90,2] + 33.649;
   1:L PR[91] R[100]mm/sec CNT100;
   1:  PR[GP1:91,1] = PR[GP1:90,1] + 41.685;
   1:  PR[GP1:91,2] = PR[GP1:90,2] + 34.382;
   1:L PR[91] R[100]mm/sec CNT100;
   1:  PR[GP1:91,1] = PR[GP1:90,1] + 36.959;
   1:  PR[GP1:91,2] = PR[GP1:90,2] + 35.375;
   1:L PR[91] R[100]mm/sec CNT100;
   1:  PR[GP1:91,1] = PR[GP1:90,1] + 30.222;
   1:  PR[GP1:91,2] = PR[GP1:90,2] + 35.572;
   1:L PR[91] R[100]mm/sec CNT100;
   1:  PR[GP1:91,1] = PR[GP1:90,1] + 23.601;
   1:  PR[GP1:91,2] = PR[GP1:90,2] + 34.701;
   1:L PR[91] R[100]mm/sec CNT100;
   1:  PR[GP1:91,1] = PR[GP1:90,1] + 17.922;
   1:  PR[GP1:91,2] = PR[GP1:90,2] + 32.894;
   1:L PR[91] R[100]mm/sec CNT100;
   1:  PR[GP1:91,1] = PR[GP1:90,1] + 16.289;
   1:  PR[GP1:91,2] = PR[GP1:90,2] + 32.328;
   1:L PR[91] R[100]mm/sec CNT100;
   1:  PR[GP1:91,1] = PR[GP1:90,1] + 11.150;
   1:  PR[GP1:91,2] = PR[GP1:90,2] + 29.646;
   1:L PR[91] R[100]mm/sec CNT100;
   1:  PR[GP1:91,1] = PR[GP1:90,1] + 10.170;
   1:  PR[GP1:91,2] = PR[GP1:90,2] + 28.954;
   1:L PR[91] R[100]mm/sec CNT100;
   1:  PR[GP1:91,1] = PR[GP1:90,1] + 6.620;
   1:  PR[GP1:91,2] = PR[GP1:90,2] + 26.176;
   1:L PR[91] R[100]mm/sec CNT100;
   1:  PR[GP1:91,1] = PR[GP1:90,1] + 3.894;
   1:  PR[GP1:91,2] = PR[GP1:90,2] + 23.004;
   1:L PR[91] R[100]mm/sec CNT100;
   1:  PR[GP1:91,1] = PR[GP1:90,1] + 3.046;
   1:  PR[GP1:91,2] = PR[GP1:90,2] + 22.669;
   1:L PR[91] R[100]mm/sec CNT100;
   1:  PR[GP1:91,1] = PR[GP1:90,1] + 0.671;
   1:  PR[GP1:91,2] = PR[GP1:90,2] + 21.455;
   1:L PR[91] R[100]mm/sec CNT100;
   1:  ! -- Layer/Ebene 74 -- !;
   1:  PR[91] = PR[90];
   1:  PR[GP1:91,1] = PR[GP1:90,1] + -1.123;
   1:  PR[GP1:91,2] = PR[GP1:90,2] + 22.021;
   1:  PR[GP1:91,3] = PR[GP1:90,3] + 45.445;
   1:L PR[91] R[100]mm/sec CNT100;
   1:  PR[GP1:91,1] = PR[GP1:90,1] + -3.664;
   1:  PR[GP1:91,2] = PR[GP1:90,2] + 23.314;
   1:L PR[91] R[100]mm/sec CNT100;
   1:  PR[GP1:91,1] = PR[GP1:90,1] + -6.219;
   1:  PR[GP1:91,2] = PR[GP1:90,2] + 26.284;
   1:L PR[91] R[100]mm/sec CNT100;
   1:  PR[GP1:91,1] = PR[GP1:90,1] + -9.613;
   1:  PR[GP1:91,2] = PR[GP1:90,2] + 28.942;
   1:L PR[91] R[100]mm/sec CNT100;
   1:  PR[GP1:91,1] = PR[GP1:90,1] + -10.710;
   1:  PR[GP1:91,2] = PR[GP1:90,2] + 29.717;
   1:L PR[91] R[100]mm/sec CNT100;
   1:  PR[GP1:91,1] = PR[GP1:90,1] + -15.743;
   1:  PR[GP1:91,2] = PR[GP1:90,2] + 32.351;
   1:L PR[91] R[100]mm/sec CNT100;
   1:  PR[GP1:91,1] = PR[GP1:90,1] + -21.907;
   1:  PR[GP1:91,2] = PR[GP1:90,2] + 34.331;
   1:L PR[91] R[100]mm/sec CNT100;
   1:  PR[GP1:91,1] = PR[GP1:90,1] + -23.202;
   1:  PR[GP1:91,2] = PR[GP1:90,2] + 34.779;
   1:L PR[91] R[100]mm/sec CNT100;
   1:  PR[GP1:91,1] = PR[GP1:90,1] + -29.670;
   1:  PR[GP1:91,2] = PR[GP1:90,2] + 35.624;
   1:L PR[91] R[100]mm/sec CNT100;
   1:  PR[GP1:91,1] = PR[GP1:90,1] + -33.891;
   1:  PR[GP1:91,2] = PR[GP1:90,2] + 35.479;
   1:L PR[91] R[100]mm/sec CNT100;
   1:  PR[GP1:91,1] = PR[GP1:90,1] + -36.656;
   1:  PR[GP1:91,2] = PR[GP1:90,2] + 35.400;
   1:L PR[91] R[100]mm/sec CNT100;
   1:  PR[GP1:91,1] = PR[GP1:90,1] + -37.660;
   1:  PR[GP1:91,2] = PR[GP1:90,2] + 35.167;
   1:L PR[91] R[100]mm/sec CNT100;
   1:  PR[GP1:91,1] = PR[GP1:90,1] + -44.226;
   1:  PR[GP1:91,2] = PR[GP1:90,2] + 33.744;
   1:L PR[91] R[100]mm/sec CNT100;
   1:  PR[GP1:91,1] = PR[GP1:90,1] + -48.468;
   1:  PR[GP1:91,2] = PR[GP1:90,2] + 32.074;
   1:L PR[91] R[100]mm/sec CNT100;
   1:  PR[GP1:91,1] = PR[GP1:90,1] + -52.590;
   1:  PR[GP1:91,2] = PR[GP1:90,2] + 29.729;
   1:L PR[91] R[100]mm/sec CNT100;
   1:  PR[GP1:91,1] = PR[GP1:90,1] + -55.745;
   1:  PR[GP1:91,2] = PR[GP1:90,2] + 27.774;
   1:L PR[91] R[100]mm/sec CNT100;
   1:  PR[GP1:91,1] = PR[GP1:90,1] + -57.791;
   1:  PR[GP1:91,2] = PR[GP1:90,2] + 25.941;
   1:L PR[91] R[100]mm/sec CNT100;
   1:  PR[GP1:91,1] = PR[GP1:90,1] + -62.462;
   1:  PR[GP1:91,2] = PR[GP1:90,2] + 21.030;
   1:L PR[91] R[100]mm/sec CNT100;
   1:  PR[GP1:91,1] = PR[GP1:90,1] + -63.722;
   1:  PR[GP1:91,2] = PR[GP1:90,2] + 19.394;
   1:L PR[91] R[100]mm/sec CNT100;
   1:  PR[GP1:91,1] = PR[GP1:90,1] + -68.054;
   1:  PR[GP1:91,2] = PR[GP1:90,2] + 10.743;
   1:L PR[91] R[100]mm/sec CNT100;
   1:  PR[GP1:91,1] = PR[GP1:90,1] + -68.419;
   1:  PR[GP1:91,2] = PR[GP1:90,2] + 9.503;
   1:L PR[91] R[100]mm/sec CNT100;
   1:  PR[GP1:91,1] = PR[GP1:90,1] + -69.752;
   1:  PR[GP1:91,2] = PR[GP1:90,2] + 0.949;
   1:L PR[91] R[100]mm/sec CNT100;
   1:  PR[GP1:91,1] = PR[GP1:90,1] + -69.842;
   1:  PR[GP1:91,2] = PR[GP1:90,2] + -0.052;
   1:L PR[91] R[100]mm/sec CNT100;
   1:  PR[GP1:91,1] = PR[GP1:90,1] + -68.527;
   1:  PR[GP1:91,2] = PR[GP1:90,2] + -8.380;
   1:L PR[91] R[100]mm/sec CNT100;
   1:  PR[GP1:91,1] = PR[GP1:90,1] + -68.413;
   1:  PR[GP1:91,2] = PR[GP1:90,2] + -9.666;
   1:L PR[91] R[100]mm/sec CNT100;
   1:  PR[GP1:91,1] = PR[GP1:90,1] + -68.054;
   1:  PR[GP1:91,2] = PR[GP1:90,2] + -10.887;
   1:L PR[91] R[100]mm/sec CNT100;
   1:  PR[GP1:91,1] = PR[GP1:90,1] + -63.722;
   1:  PR[GP1:91,2] = PR[GP1:90,2] + -19.538;
   1:L PR[91] R[100]mm/sec CNT100;
   1:  PR[GP1:91,1] = PR[GP1:90,1] + -62.462;
   1:  PR[GP1:91,2] = PR[GP1:90,2] + -21.174;
   1:L PR[91] R[100]mm/sec CNT100;
   1:  PR[GP1:91,1] = PR[GP1:90,1] + -57.790;
   1:  PR[GP1:91,2] = PR[GP1:90,2] + -26.085;
   1:L PR[91] R[100]mm/sec CNT100;
   1:  PR[GP1:91,1] = PR[GP1:90,1] + -55.755;
   1:  PR[GP1:91,2] = PR[GP1:90,2] + -27.910;
   1:L PR[91] R[100]mm/sec CNT100;
   1:  PR[GP1:91,1] = PR[GP1:90,1] + -51.368;
   1:  PR[GP1:91,2] = PR[GP1:90,2] + -30.378;
   1:L PR[91] R[100]mm/sec CNT100;
   1:  PR[GP1:91,1] = PR[GP1:90,1] + -48.454;
   1:  PR[GP1:91,2] = PR[GP1:90,2] + -32.224;
   1:L PR[91] R[100]mm/sec CNT100;
   1:  PR[GP1:91,1] = PR[GP1:90,1] + -44.221;
   1:  PR[GP1:91,2] = PR[GP1:90,2] + -33.890;
   1:L PR[91] R[100]mm/sec CNT100;
   1:  PR[GP1:91,1] = PR[GP1:90,1] + -41.741;
   1:  PR[GP1:91,2] = PR[GP1:90,2] + -34.473;
   1:L PR[91] R[100]mm/sec CNT100;
   1:  PR[GP1:91,1] = PR[GP1:90,1] + -36.663;
   1:  PR[GP1:91,2] = PR[GP1:90,2] + -35.544;
   1:L PR[91] R[100]mm/sec CNT100;
   1:  PR[GP1:91,1] = PR[GP1:90,1] + -33.890;
   1:  PR[GP1:91,2] = PR[GP1:90,2] + -35.623;
   1:L PR[91] R[100]mm/sec CNT100;
   1:  PR[GP1:91,1] = PR[GP1:90,1] + -30.133;
   1:  PR[GP1:91,2] = PR[GP1:90,2] + -35.767;
   1:L PR[91] R[100]mm/sec CNT100;
   1:  PR[GP1:91,1] = PR[GP1:90,1] + -29.679;
   1:  PR[GP1:91,2] = PR[GP1:90,2] + -35.769;
   1:L PR[91] R[100]mm/sec CNT100;
   1:  PR[GP1:91,1] = PR[GP1:90,1] + -23.193;
   1:  PR[GP1:91,2] = PR[GP1:90,2] + -34.921;
   1:L PR[91] R[100]mm/sec CNT100;
   1:  PR[GP1:91,1] = PR[GP1:90,1] + -17.651;
   1:  PR[GP1:91,2] = PR[GP1:90,2] + -33.158;
   1:L PR[91] R[100]mm/sec CNT100;
   1:  PR[GP1:91,1] = PR[GP1:90,1] + -15.747;
   1:  PR[GP1:91,2] = PR[GP1:90,2] + -32.496;
   1:L PR[91] R[100]mm/sec CNT100;
   1:  PR[GP1:91,1] = PR[GP1:90,1] + -10.711;
   1:  PR[GP1:91,2] = PR[GP1:90,2] + -29.861;
   1:L PR[91] R[100]mm/sec CNT100;
   1:  PR[GP1:91,1] = PR[GP1:90,1] + -9.187;
   1:  PR[GP1:91,2] = PR[GP1:90,2] + -28.754;
   1:L PR[91] R[100]mm/sec CNT100;
   1:  PR[GP1:91,1] = PR[GP1:90,1] + -6.014;
   1:  PR[GP1:91,2] = PR[GP1:90,2] + -26.269;
   1:L PR[91] R[100]mm/sec CNT100;
   1:  PR[GP1:91,1] = PR[GP1:90,1] + -3.608;
   1:  PR[GP1:91,2] = PR[GP1:90,2] + -23.479;
   1:L PR[91] R[100]mm/sec CNT100;
   1:  PR[GP1:91,1] = PR[GP1:90,1] + -1.634;
   1:  PR[GP1:91,2] = PR[GP1:90,2] + -23.055;
   1:L PR[91] R[100]mm/sec CNT100;
   1:  PR[GP1:91,1] = PR[GP1:90,1] + 0.599;
   1:  PR[GP1:91,2] = PR[GP1:90,2] + -21.872;
   1:L PR[91] R[100]mm/sec CNT100;
   1:  PR[GP1:91,1] = PR[GP1:90,1] + 3.882;
   1:  PR[GP1:91,2] = PR[GP1:90,2] + -23.542;
   1:L PR[91] R[100]mm/sec CNT100;
   1:  PR[GP1:91,1] = PR[GP1:90,1] + 6.255;
   1:  PR[GP1:91,2] = PR[GP1:90,2] + -26.297;
   1:L PR[91] R[100]mm/sec CNT100;
   1:  PR[GP1:91,1] = PR[GP1:90,1] + 9.413;
   1:  PR[GP1:91,2] = PR[GP1:90,2] + -28.768;
   1:L PR[91] R[100]mm/sec CNT100;
   1:  PR[GP1:91,1] = PR[GP1:90,1] + 10.940;
   1:  PR[GP1:91,2] = PR[GP1:90,2] + -29.878;
   1:L PR[91] R[100]mm/sec CNT100;
   1:  PR[GP1:91,1] = PR[GP1:90,1] + 15.938;
   1:  PR[GP1:91,2] = PR[GP1:90,2] + -32.486;
   1:L PR[91] R[100]mm/sec CNT100;
   1:  PR[GP1:91,1] = PR[GP1:90,1] + 22.110;
   1:  PR[GP1:91,2] = PR[GP1:90,2] + -34.469;
   1:L PR[91] R[100]mm/sec CNT100;
   1:  PR[GP1:91,1] = PR[GP1:90,1] + 23.408;
   1:  PR[GP1:91,2] = PR[GP1:90,2] + -34.918;
   1:L PR[91] R[100]mm/sec CNT100;
   1:  PR[GP1:91,1] = PR[GP1:90,1] + 29.869;
   1:  PR[GP1:91,2] = PR[GP1:90,2] + -35.768;
   1:L PR[91] R[100]mm/sec CNT100;
   1:  PR[GP1:91,1] = PR[GP1:90,1] + 36.829;
   1:  PR[GP1:91,2] = PR[GP1:90,2] + -35.550;
   1:L PR[91] R[100]mm/sec CNT100;
   1:  PR[GP1:91,1] = PR[GP1:90,1] + 37.821;
   1:  PR[GP1:91,2] = PR[GP1:90,2] + -35.319;
   1:L PR[91] R[100]mm/sec CNT100;
   1:  PR[GP1:91,1] = PR[GP1:90,1] + 44.401;
   1:  PR[GP1:91,2] = PR[GP1:90,2] + -33.896;
   1:L PR[91] R[100]mm/sec CNT100;
   1:  PR[GP1:91,1] = PR[GP1:90,1] + 48.661;
   1:  PR[GP1:91,2] = PR[GP1:90,2] + -32.228;
   1:L PR[91] R[100]mm/sec CNT100;
   1:  PR[GP1:91,1] = PR[GP1:90,1] + 52.781;
   1:  PR[GP1:91,2] = PR[GP1:90,2] + -29.888;
   1:L PR[91] R[100]mm/sec CNT100;
   1:  PR[GP1:91,1] = PR[GP1:90,1] + 55.928;
   1:  PR[GP1:91,2] = PR[GP1:90,2] + -27.947;
   1:L PR[91] R[100]mm/sec CNT100;
   1:  PR[GP1:91,1] = PR[GP1:90,1] + 57.972;
   1:  PR[GP1:91,2] = PR[GP1:90,2] + -26.121;
   1:L PR[91] R[100]mm/sec CNT100;
   1:  PR[GP1:91,1] = PR[GP1:90,1] + 62.644;
   1:  PR[GP1:91,2] = PR[GP1:90,2] + -21.193;
   1:L PR[91] R[100]mm/sec CNT100;
   1:  PR[GP1:91,1] = PR[GP1:90,1] + 63.924;
   1:  PR[GP1:91,2] = PR[GP1:90,2] + -19.537;
   1:L PR[91] R[100]mm/sec CNT100;
   1:  PR[GP1:91,1] = PR[GP1:90,1] + 68.261;
   1:  PR[GP1:91,2] = PR[GP1:90,2] + -10.928;
   1:L PR[91] R[100]mm/sec CNT100;
   1:  PR[GP1:91,1] = PR[GP1:90,1] + 68.626;
   1:  PR[GP1:91,2] = PR[GP1:90,2] + -9.706;
   1:L PR[91] R[100]mm/sec CNT100;
   1:  PR[GP1:91,1] = PR[GP1:90,1] + 69.961;
   1:  PR[GP1:91,2] = PR[GP1:90,2] + -1.123;
   1:L PR[91] R[100]mm/sec CNT100;
   1:  PR[GP1:91,1] = PR[GP1:90,1] + 70.056;
   1:  PR[GP1:91,2] = PR[GP1:90,2] + -0.092;
   1:L PR[91] R[100]mm/sec CNT100;
   1:  PR[GP1:91,1] = PR[GP1:90,1] + 68.740;
   1:  PR[GP1:91,2] = PR[GP1:90,2] + 8.259;
   1:L PR[91] R[100]mm/sec CNT100;
   1:  PR[GP1:91,1] = PR[GP1:90,1] + 68.621;
   1:  PR[GP1:91,2] = PR[GP1:90,2] + 9.580;
   1:L PR[91] R[100]mm/sec CNT100;
   1:  PR[GP1:91,1] = PR[GP1:90,1] + 68.261;
   1:  PR[GP1:91,2] = PR[GP1:90,2] + 10.785;
   1:L PR[91] R[100]mm/sec CNT100;
   1:  PR[GP1:91,1] = PR[GP1:90,1] + 64.758;
   1:  PR[GP1:91,2] = PR[GP1:90,2] + 17.763;
   1:L PR[91] R[100]mm/sec CNT100;
   1:  PR[GP1:91,1] = PR[GP1:90,1] + 63.925;
   1:  PR[GP1:91,2] = PR[GP1:90,2] + 19.392;
   1:L PR[91] R[100]mm/sec CNT100;
   1:  PR[GP1:91,1] = PR[GP1:90,1] + 62.644;
   1:  PR[GP1:91,2] = PR[GP1:90,2] + 21.049;
   1:L PR[91] R[100]mm/sec CNT100;
   1:  PR[GP1:91,1] = PR[GP1:90,1] + 57.972;
   1:  PR[GP1:91,2] = PR[GP1:90,2] + 25.977;
   1:L PR[91] R[100]mm/sec CNT100;
   1:  PR[GP1:91,1] = PR[GP1:90,1] + 55.938;
   1:  PR[GP1:91,2] = PR[GP1:90,2] + 27.795;
   1:L PR[91] R[100]mm/sec CNT100;
   1:  PR[GP1:91,1] = PR[GP1:90,1] + 51.553;
   1:  PR[GP1:91,2] = PR[GP1:90,2] + 30.258;
   1:L PR[91] R[100]mm/sec CNT100;
   1:  PR[GP1:91,1] = PR[GP1:90,1] + 48.648;
   1:  PR[GP1:91,2] = PR[GP1:90,2] + 32.089;
   1:L PR[91] R[100]mm/sec CNT100;
   1:  PR[GP1:91,1] = PR[GP1:90,1] + 44.396;
   1:  PR[GP1:91,2] = PR[GP1:90,2] + 33.754;
   1:L PR[91] R[100]mm/sec CNT100;
   1:  PR[GP1:91,1] = PR[GP1:90,1] + 41.923;
   1:  PR[GP1:91,2] = PR[GP1:90,2] + 34.337;
   1:L PR[91] R[100]mm/sec CNT100;
   1:  PR[GP1:91,1] = PR[GP1:90,1] + 36.837;
   1:  PR[GP1:91,2] = PR[GP1:90,2] + 35.405;
   1:L PR[91] R[100]mm/sec CNT100;
   1:  PR[GP1:91,1] = PR[GP1:90,1] + 34.103;
   1:  PR[GP1:91,2] = PR[GP1:90,2] + 35.481;
   1:L PR[91] R[100]mm/sec CNT100;
   1:  PR[GP1:91,1] = PR[GP1:90,1] + 30.334;
   1:  PR[GP1:91,2] = PR[GP1:90,2] + 35.623;
   1:L PR[91] R[100]mm/sec CNT100;
   1:  PR[GP1:91,1] = PR[GP1:90,1] + 29.878;
   1:  PR[GP1:91,2] = PR[GP1:90,2] + 35.625;
   1:L PR[91] R[100]mm/sec CNT100;
   1:  PR[GP1:91,1] = PR[GP1:90,1] + 23.403;
   1:  PR[GP1:91,2] = PR[GP1:90,2] + 34.774;
   1:L PR[91] R[100]mm/sec CNT100;
   1:  PR[GP1:91,1] = PR[GP1:90,1] + 17.855;
   1:  PR[GP1:91,2] = PR[GP1:90,2] + 33.008;
   1:L PR[91] R[100]mm/sec CNT100;
   1:  PR[GP1:91,1] = PR[GP1:90,1] + 15.948;
   1:  PR[GP1:91,2] = PR[GP1:90,2] + 32.347;
   1:L PR[91] R[100]mm/sec CNT100;
   1:  PR[GP1:91,1] = PR[GP1:90,1] + 10.939;
   1:  PR[GP1:91,2] = PR[GP1:90,2] + 29.733;
   1:L PR[91] R[100]mm/sec CNT100;
   1:  PR[GP1:91,1] = PR[GP1:90,1] + 9.839;
   1:  PR[GP1:91,2] = PR[GP1:90,2] + 28.957;
   1:L PR[91] R[100]mm/sec CNT100;
   1:  PR[GP1:91,1] = PR[GP1:90,1] + 6.462;
   1:  PR[GP1:91,2] = PR[GP1:90,2] + 26.314;
   1:L PR[91] R[100]mm/sec CNT100;
   1:  PR[GP1:91,1] = PR[GP1:90,1] + 3.864;
   1:  PR[GP1:91,2] = PR[GP1:90,2] + 23.291;
   1:L PR[91] R[100]mm/sec CNT100;
   1:  PR[GP1:91,1] = PR[GP1:90,1] + 2.957;
   1:  PR[GP1:91,2] = PR[GP1:90,2] + 22.932;
   1:L PR[91] R[100]mm/sec CNT100;
   1:  PR[GP1:91,1] = PR[GP1:90,1] + 0.712;
   1:  PR[GP1:91,2] = PR[GP1:90,2] + 21.785;
   1:L PR[91] R[100]mm/sec CNT100;
   1:  ! -- Layer/Ebene 75 -- !;
   1:  PR[91] = PR[90];
   1:  PR[GP1:91,1] = PR[GP1:90,1] + -1.212;
   1:  PR[GP1:91,2] = PR[GP1:90,2] + 22.367;
   1:  PR[GP1:91,3] = PR[GP1:90,3] + 46.055;
   1:L PR[91] R[100]mm/sec CNT100;
   1:  PR[GP1:91,1] = PR[GP1:90,1] + -3.635;
   1:  PR[GP1:91,2] = PR[GP1:90,2] + 23.600;
   1:L PR[91] R[100]mm/sec CNT100;
   1:  PR[GP1:91,1] = PR[GP1:90,1] + -6.063;
   1:  PR[GP1:91,2] = PR[GP1:90,2] + 26.423;
   1:L PR[91] R[100]mm/sec CNT100;
   1:  PR[GP1:91,1] = PR[GP1:90,1] + -9.283;
   1:  PR[GP1:91,2] = PR[GP1:90,2] + 28.945;
   1:L PR[91] R[100]mm/sec CNT100;
   1:  PR[GP1:91,1] = PR[GP1:90,1] + -10.499;
   1:  PR[GP1:91,2] = PR[GP1:90,2] + 29.804;
   1:L PR[91] R[100]mm/sec CNT100;
   1:  PR[GP1:91,1] = PR[GP1:90,1] + -15.402;
   1:  PR[GP1:91,2] = PR[GP1:90,2] + 32.369;
   1:L PR[91] R[100]mm/sec CNT100;
   1:  PR[GP1:91,1] = PR[GP1:90,1] + -21.406;
   1:  PR[GP1:91,2] = PR[GP1:90,2] + 34.298;
   1:L PR[91] R[100]mm/sec CNT100;
   1:  PR[GP1:91,1] = PR[GP1:90,1] + -23.004;
   1:  PR[GP1:91,2] = PR[GP1:90,2] + 34.851;
   1:L PR[91] R[100]mm/sec CNT100;
   1:  PR[GP1:91,1] = PR[GP1:90,1] + -29.319;
   1:  PR[GP1:91,2] = PR[GP1:90,2] + 35.676;
   1:L PR[91] R[100]mm/sec CNT100;
   1:  PR[GP1:91,1] = PR[GP1:90,1] + -36.539;
   1:  PR[GP1:91,2] = PR[GP1:90,2] + 35.431;
   1:L PR[91] R[100]mm/sec CNT100;
   1:  PR[GP1:91,1] = PR[GP1:90,1] + -43.832;
   1:  PR[GP1:91,2] = PR[GP1:90,2] + 33.848;
   1:L PR[91] R[100]mm/sec CNT100;
   1:  PR[GP1:91,1] = PR[GP1:90,1] + -48.472;
   1:  PR[GP1:91,2] = PR[GP1:90,2] + 32.021;
   1:L PR[91] R[100]mm/sec CNT100;
   1:  PR[GP1:91,1] = PR[GP1:90,1] + -51.966;
   1:  PR[GP1:91,2] = PR[GP1:90,2] + 30.033;
   1:L PR[91] R[100]mm/sec CNT100;
   1:  PR[GP1:91,1] = PR[GP1:90,1] + -55.532;
   1:  PR[GP1:91,2] = PR[GP1:90,2] + 27.824;
   1:L PR[91] R[100]mm/sec CNT100;
   1:  PR[GP1:91,1] = PR[GP1:90,1] + -57.846;
   1:  PR[GP1:91,2] = PR[GP1:90,2] + 25.750;
   1:L PR[91] R[100]mm/sec CNT100;
   1:  PR[GP1:91,1] = PR[GP1:90,1] + -62.095;
   1:  PR[GP1:91,2] = PR[GP1:90,2] + 21.283;
   1:L PR[91] R[100]mm/sec CNT100;
   1:  PR[GP1:91,1] = PR[GP1:90,1] + -63.597;
   1:  PR[GP1:91,2] = PR[GP1:90,2] + 19.333;
   1:L PR[91] R[100]mm/sec CNT100;
   1:  PR[GP1:91,1] = PR[GP1:90,1] + -67.837;
   1:  PR[GP1:91,2] = PR[GP1:90,2] + 10.870;
   1:L PR[91] R[100]mm/sec CNT100;
   1:  PR[GP1:91,1] = PR[GP1:90,1] + -68.302;
   1:  PR[GP1:91,2] = PR[GP1:90,2] + 9.289;
   1:L PR[91] R[100]mm/sec CNT100;
   1:  PR[GP1:91,1] = PR[GP1:90,1] + -69.546;
   1:  PR[GP1:91,2] = PR[GP1:90,2] + 1.312;
   1:L PR[91] R[100]mm/sec CNT100;
   1:  PR[GP1:91,1] = PR[GP1:90,1] + -69.668;
   1:  PR[GP1:91,2] = PR[GP1:90,2] + -0.052;
   1:L PR[91] R[100]mm/sec CNT100;
   1:  PR[GP1:91,1] = PR[GP1:90,1] + -68.440;
   1:  PR[GP1:91,2] = PR[GP1:90,2] + -7.827;
   1:L PR[91] R[100]mm/sec CNT100;
   1:  PR[GP1:91,1] = PR[GP1:90,1] + -68.297;
   1:  PR[GP1:91,2] = PR[GP1:90,2] + -9.452;
   1:L PR[91] R[100]mm/sec CNT100;
   1:  PR[GP1:91,1] = PR[GP1:90,1] + -67.837;
   1:  PR[GP1:91,2] = PR[GP1:90,2] + -11.014;
   1:L PR[91] R[100]mm/sec CNT100;
   1:  PR[GP1:91,1] = PR[GP1:90,1] + -63.597;
   1:  PR[GP1:91,2] = PR[GP1:90,2] + -19.477;
   1:L PR[91] R[100]mm/sec CNT100;
   1:  PR[GP1:91,1] = PR[GP1:90,1] + -62.095;
   1:  PR[GP1:91,2] = PR[GP1:90,2] + -21.427;
   1:L PR[91] R[100]mm/sec CNT100;
   1:  PR[GP1:91,1] = PR[GP1:90,1] + -57.846;
   1:  PR[GP1:91,2] = PR[GP1:90,2] + -25.894;
   1:L PR[91] R[100]mm/sec CNT100;
   1:  PR[GP1:91,1] = PR[GP1:90,1] + -55.542;
   1:  PR[GP1:91,2] = PR[GP1:90,2] + -27.960;
   1:L PR[91] R[100]mm/sec CNT100;
   1:  PR[GP1:91,1] = PR[GP1:90,1] + -51.644;
   1:  PR[GP1:91,2] = PR[GP1:90,2] + -30.152;
   1:L PR[91] R[100]mm/sec CNT100;
   1:  PR[GP1:91,1] = PR[GP1:90,1] + -48.459;
   1:  PR[GP1:91,2] = PR[GP1:90,2] + -32.171;
   1:L PR[91] R[100]mm/sec CNT100;
   1:  PR[GP1:91,1] = PR[GP1:90,1] + -43.827;
   1:  PR[GP1:91,2] = PR[GP1:90,2] + -33.993;
   1:L PR[91] R[100]mm/sec CNT100;
   1:  PR[GP1:91,1] = PR[GP1:90,1] + -41.981;
   1:  PR[GP1:91,2] = PR[GP1:90,2] + -34.428;
   1:L PR[91] R[100]mm/sec CNT100;
   1:  PR[GP1:91,1] = PR[GP1:90,1] + -36.540;
   1:  PR[GP1:91,2] = PR[GP1:90,2] + -35.575;
   1:L PR[91] R[100]mm/sec CNT100;
   1:  PR[GP1:91,1] = PR[GP1:90,1] + -30.088;
   1:  PR[GP1:91,2] = PR[GP1:90,2] + -35.819;
   1:L PR[91] R[100]mm/sec CNT100;
   1:  PR[GP1:91,1] = PR[GP1:90,1] + -29.327;
   1:  PR[GP1:91,2] = PR[GP1:90,2] + -35.821;
   1:L PR[91] R[100]mm/sec CNT100;
   1:  PR[GP1:91,1] = PR[GP1:90,1] + -22.994;
   1:  PR[GP1:91,2] = PR[GP1:90,2] + -34.993;
   1:L PR[91] R[100]mm/sec CNT100;
   1:  PR[GP1:91,1] = PR[GP1:90,1] + -17.583;
   1:  PR[GP1:91,2] = PR[GP1:90,2] + -33.271;
   1:L PR[91] R[100]mm/sec CNT100;
   1:  PR[GP1:91,1] = PR[GP1:90,1] + -15.404;
   1:  PR[GP1:91,2] = PR[GP1:90,2] + -32.514;
   1:L PR[91] R[100]mm/sec CNT100;
   1:  PR[GP1:91,1] = PR[GP1:90,1] + -10.500;
   1:  PR[GP1:91,2] = PR[GP1:90,2] + -29.948;
   1:L PR[91] R[100]mm/sec CNT100;
   1:  PR[GP1:91,1] = PR[GP1:90,1] + -8.812;
   1:  PR[GP1:91,2] = PR[GP1:90,2] + -28.722;
   1:L PR[91] R[100]mm/sec CNT100;
   1:  PR[GP1:91,1] = PR[GP1:90,1] + -5.841;
   1:  PR[GP1:91,2] = PR[GP1:90,2] + -26.395;
   1:L PR[91] R[100]mm/sec CNT100;
   1:  PR[GP1:91,1] = PR[GP1:90,1] + -3.579;
   1:  PR[GP1:91,2] = PR[GP1:90,2] + -23.772;
   1:L PR[91] R[100]mm/sec CNT100;
   1:  PR[GP1:91,1] = PR[GP1:90,1] + -1.467;
   1:  PR[GP1:91,2] = PR[GP1:90,2] + -23.319;
   1:L PR[91] R[100]mm/sec CNT100;
   1:  PR[GP1:91,1] = PR[GP1:90,1] + 0.640;
   1:  PR[GP1:91,2] = PR[GP1:90,2] + -22.202;
   1:L PR[91] R[100]mm/sec CNT100;
   1:  PR[GP1:91,1] = PR[GP1:90,1] + 3.852;
   1:  PR[GP1:91,2] = PR[GP1:90,2] + -23.835;
   1:L PR[91] R[100]mm/sec CNT100;
   1:  PR[GP1:91,1] = PR[GP1:90,1] + 6.080;
   1:  PR[GP1:91,2] = PR[GP1:90,2] + -26.422;
   1:L PR[91] R[100]mm/sec CNT100;
   1:  PR[GP1:91,1] = PR[GP1:90,1] + 9.038;
   1:  PR[GP1:91,2] = PR[GP1:90,2] + -28.736;
   1:L PR[91] R[100]mm/sec CNT100;
   1:  PR[GP1:91,1] = PR[GP1:90,1] + 10.728;
   1:  PR[GP1:91,2] = PR[GP1:90,2] + -29.964;
   1:L PR[91] R[100]mm/sec CNT100;
   1:  PR[GP1:91,1] = PR[GP1:90,1] + 15.596;
   1:  PR[GP1:91,2] = PR[GP1:90,2] + -32.505;
   1:L PR[91] R[100]mm/sec CNT100;
   1:  PR[GP1:91,1] = PR[GP1:90,1] + 21.609;
   1:  PR[GP1:91,2] = PR[GP1:90,2] + -34.436;
   1:L PR[91] R[100]mm/sec CNT100;
   1:  PR[GP1:91,1] = PR[GP1:90,1] + 23.210;
   1:  PR[GP1:91,2] = PR[GP1:90,2] + -34.991;
   1:L PR[91] R[100]mm/sec CNT100;
   1:  PR[GP1:91,1] = PR[GP1:90,1] + 29.517;
   1:  PR[GP1:91,2] = PR[GP1:90,2] + -35.820;
   1:L PR[91] R[100]mm/sec CNT100;
   1:  PR[GP1:91,1] = PR[GP1:90,1] + 36.711;
   1:  PR[GP1:91,2] = PR[GP1:90,2] + -35.580;
   1:L PR[91] R[100]mm/sec CNT100;
   1:  PR[GP1:91,1] = PR[GP1:90,1] + 44.003;
   1:  PR[GP1:91,2] = PR[GP1:90,2] + -34.000;
   1:L PR[91] R[100]mm/sec CNT100;
   1:  PR[GP1:91,1] = PR[GP1:90,1] + 48.664;
   1:  PR[GP1:91,2] = PR[GP1:90,2] + -32.176;
   1:L PR[91] R[100]mm/sec CNT100;
   1:  PR[GP1:91,1] = PR[GP1:90,1] + 52.154;
   1:  PR[GP1:91,2] = PR[GP1:90,2] + -30.193;
   1:L PR[91] R[100]mm/sec CNT100;
   1:  PR[GP1:91,1] = PR[GP1:90,1] + 55.711;
   1:  PR[GP1:91,2] = PR[GP1:90,2] + -28.000;
   1:L PR[91] R[100]mm/sec CNT100;
   1:  PR[GP1:91,1] = PR[GP1:90,1] + 58.023;
   1:  PR[GP1:91,2] = PR[GP1:90,2] + -25.934;
   1:L PR[91] R[100]mm/sec CNT100;
   1:  PR[GP1:91,1] = PR[GP1:90,1] + 62.272;
   1:  PR[GP1:91,2] = PR[GP1:90,2] + -21.453;
   1:L PR[91] R[100]mm/sec CNT100;
   1:  PR[GP1:91,1] = PR[GP1:90,1] + 63.797;
   1:  PR[GP1:91,2] = PR[GP1:90,2] + -19.479;
   1:L PR[91] R[100]mm/sec CNT100;
   1:  PR[GP1:91,1] = PR[GP1:90,1] + 67.125;
   1:  PR[GP1:91,2] = PR[GP1:90,2] + -12.857;
   1:L PR[91] R[100]mm/sec CNT100;
   1:  PR[GP1:91,1] = PR[GP1:90,1] + 68.043;
   1:  PR[GP1:91,2] = PR[GP1:90,2] + -11.057;
   1:L PR[91] R[100]mm/sec CNT100;
   1:  PR[GP1:91,1] = PR[GP1:90,1] + 68.508;
   1:  PR[GP1:91,2] = PR[GP1:90,2] + -9.499;
   1:L PR[91] R[100]mm/sec CNT100;
   1:  PR[GP1:91,1] = PR[GP1:90,1] + 69.753;
   1:  PR[GP1:91,2] = PR[GP1:90,2] + -1.497;
   1:L PR[91] R[100]mm/sec CNT100;
   1:  PR[GP1:91,1] = PR[GP1:90,1] + 69.882;
   1:  PR[GP1:91,2] = PR[GP1:90,2] + -0.092;
   1:L PR[91] R[100]mm/sec CNT100;
   1:  PR[GP1:91,1] = PR[GP1:90,1] + 68.653;
   1:  PR[GP1:91,2] = PR[GP1:90,2] + 7.704;
   1:L PR[91] R[100]mm/sec CNT100;
   1:  PR[GP1:91,1] = PR[GP1:90,1] + 68.503;
   1:  PR[GP1:91,2] = PR[GP1:90,2] + 9.374;
   1:L PR[91] R[100]mm/sec CNT100;
   1:  PR[GP1:91,1] = PR[GP1:90,1] + 68.043;
   1:  PR[GP1:91,2] = PR[GP1:90,2] + 10.915;
   1:L PR[91] R[100]mm/sec CNT100;
   1:  PR[GP1:91,1] = PR[GP1:90,1] + 64.788;
   1:  PR[GP1:91,2] = PR[GP1:90,2] + 17.397;
   1:L PR[91] R[100]mm/sec CNT100;
   1:  PR[GP1:91,1] = PR[GP1:90,1] + 63.798;
   1:  PR[GP1:91,2] = PR[GP1:90,2] + 19.334;
   1:L PR[91] R[100]mm/sec CNT100;
   1:  PR[GP1:91,1] = PR[GP1:90,1] + 62.272;
   1:  PR[GP1:91,2] = PR[GP1:90,2] + 21.309;
   1:L PR[91] R[100]mm/sec CNT100;
   1:  PR[GP1:91,1] = PR[GP1:90,1] + 58.023;
   1:  PR[GP1:91,2] = PR[GP1:90,2] + 25.790;
   1:L PR[91] R[100]mm/sec CNT100;
   1:  PR[GP1:91,1] = PR[GP1:90,1] + 55.720;
   1:  PR[GP1:91,2] = PR[GP1:90,2] + 27.848;
   1:L PR[91] R[100]mm/sec CNT100;
   1:  PR[GP1:91,1] = PR[GP1:90,1] + 51.826;
   1:  PR[GP1:91,2] = PR[GP1:90,2] + 30.036;
   1:L PR[91] R[100]mm/sec CNT100;
   1:  PR[GP1:91,1] = PR[GP1:90,1] + 48.651;
   1:  PR[GP1:91,2] = PR[GP1:90,2] + 32.037;
   1:L PR[91] R[100]mm/sec CNT100;
   1:  PR[GP1:91,1] = PR[GP1:90,1] + 43.998;
   1:  PR[GP1:91,2] = PR[GP1:90,2] + 33.858;
   1:L PR[91] R[100]mm/sec CNT100;
   1:  PR[GP1:91,1] = PR[GP1:90,1] + 42.161;
   1:  PR[GP1:91,2] = PR[GP1:90,2] + 34.292;
   1:L PR[91] R[100]mm/sec CNT100;
   1:  PR[GP1:91,1] = PR[GP1:90,1] + 36.712;
   1:  PR[GP1:91,2] = PR[GP1:90,2] + 35.437;
   1:L PR[91] R[100]mm/sec CNT100;
   1:  PR[GP1:91,1] = PR[GP1:90,1] + 30.289;
   1:  PR[GP1:91,2] = PR[GP1:90,2] + 35.675;
   1:L PR[91] R[100]mm/sec CNT100;
   1:  PR[GP1:91,1] = PR[GP1:90,1] + 29.527;
   1:  PR[GP1:91,2] = PR[GP1:90,2] + 35.677;
   1:L PR[91] R[100]mm/sec CNT100;
   1:  PR[GP1:91,1] = PR[GP1:90,1] + 23.204;
   1:  PR[GP1:91,2] = PR[GP1:90,2] + 34.846;
   1:L PR[91] R[100]mm/sec CNT100;
   1:  PR[GP1:91,1] = PR[GP1:90,1] + 17.787;
   1:  PR[GP1:91,2] = PR[GP1:90,2] + 33.122;
   1:L PR[91] R[100]mm/sec CNT100;
   1:  PR[GP1:91,1] = PR[GP1:90,1] + 15.606;
   1:  PR[GP1:91,2] = PR[GP1:90,2] + 32.366;
   1:L PR[91] R[100]mm/sec CNT100;
   1:  PR[GP1:91,1] = PR[GP1:90,1] + 10.727;
   1:  PR[GP1:91,2] = PR[GP1:90,2] + 29.820;
   1:L PR[91] R[100]mm/sec CNT100;
   1:  PR[GP1:91,1] = PR[GP1:90,1] + 9.509;
   1:  PR[GP1:91,2] = PR[GP1:90,2] + 28.959;
   1:L PR[91] R[100]mm/sec CNT100;
   1:  PR[GP1:91,1] = PR[GP1:90,1] + 6.304;
   1:  PR[GP1:91,2] = PR[GP1:90,2] + 26.452;
   1:L PR[91] R[100]mm/sec CNT100;
   1:  PR[GP1:91,1] = PR[GP1:90,1] + 3.834;
   1:  PR[GP1:91,2] = PR[GP1:90,2] + 23.577;
   1:L PR[91] R[100]mm/sec CNT100;
   1:  PR[GP1:91,1] = PR[GP1:90,1] + 2.868;
   1:  PR[GP1:91,2] = PR[GP1:90,2] + 23.196;
   1:L PR[91] R[100]mm/sec CNT100;
   1:  PR[GP1:91,1] = PR[GP1:90,1] + 0.754;
   1:  PR[GP1:91,2] = PR[GP1:90,2] + 22.115;
   1:L PR[91] R[100]mm/sec CNT100;
   1:  ! -- Layer/Ebene 76 -- !;
   1:  PR[91] = PR[90];
   1:  PR[GP1:91,1] = PR[GP1:90,1] + -1.300;
   1:  PR[GP1:91,2] = PR[GP1:90,2] + 22.714;
   1:  PR[GP1:91,3] = PR[GP1:90,3] + 46.665;
   1:L PR[91] R[100]mm/sec CNT100;
   1:  PR[GP1:91,1] = PR[GP1:90,1] + -3.606;
   1:  PR[GP1:91,2] = PR[GP1:90,2] + 23.887;
   1:L PR[91] R[100]mm/sec CNT100;
   1:  PR[GP1:91,1] = PR[GP1:90,1] + -5.907;
   1:  PR[GP1:91,2] = PR[GP1:90,2] + 26.563;
   1:L PR[91] R[100]mm/sec CNT100;
   1:  PR[GP1:91,1] = PR[GP1:90,1] + -8.954;
   1:  PR[GP1:91,2] = PR[GP1:90,2] + 28.948;
   1:L PR[91] R[100]mm/sec CNT100;
   1:  PR[GP1:91,1] = PR[GP1:90,1] + -10.288;
   1:  PR[GP1:91,2] = PR[GP1:90,2] + 29.892;
   1:L PR[91] R[100]mm/sec CNT100;
   1:  PR[GP1:91,1] = PR[GP1:90,1] + -15.060;
   1:  PR[GP1:91,2] = PR[GP1:90,2] + 32.388;
   1:L PR[91] R[100]mm/sec CNT100;
   1:  PR[GP1:91,1] = PR[GP1:90,1] + -20.905;
   1:  PR[GP1:91,2] = PR[GP1:90,2] + 34.266;
   1:L PR[91] R[100]mm/sec CNT100;
   1:  PR[GP1:91,1] = PR[GP1:90,1] + -22.805;
   1:  PR[GP1:91,2] = PR[GP1:90,2] + 34.923;
   1:L PR[91] R[100]mm/sec CNT100;
   1:  PR[GP1:91,1] = PR[GP1:90,1] + -28.968;
   1:  PR[GP1:91,2] = PR[GP1:90,2] + 35.728;
   1:L PR[91] R[100]mm/sec CNT100;
   1:  PR[GP1:91,1] = PR[GP1:90,1] + -36.365;
   1:  PR[GP1:91,2] = PR[GP1:90,2] + 35.482;
   1:L PR[91] R[100]mm/sec CNT100;
   1:  PR[GP1:91,1] = PR[GP1:90,1] + -43.438;
   1:  PR[GP1:91,2] = PR[GP1:90,2] + 33.951;
   1:L PR[91] R[100]mm/sec CNT100;
   1:  PR[GP1:91,1] = PR[GP1:90,1] + -48.476;
   1:  PR[GP1:91,2] = PR[GP1:90,2] + 31.968;
   1:L PR[91] R[100]mm/sec CNT100;
   1:  PR[GP1:91,1] = PR[GP1:90,1] + -51.342;
   1:  PR[GP1:91,2] = PR[GP1:90,2] + 30.338;
   1:L PR[91] R[100]mm/sec CNT100;
   1:  PR[GP1:91,1] = PR[GP1:90,1] + -55.319;
   1:  PR[GP1:91,2] = PR[GP1:90,2] + 27.874;
   1:L PR[91] R[100]mm/sec CNT100;
   1:  PR[GP1:91,1] = PR[GP1:90,1] + -57.902;
   1:  PR[GP1:91,2] = PR[GP1:90,2] + 25.558;
   1:L PR[91] R[100]mm/sec CNT100;
   1:  PR[GP1:91,1] = PR[GP1:90,1] + -61.728;
   1:  PR[GP1:91,2] = PR[GP1:90,2] + 21.536;
   1:L PR[91] R[100]mm/sec CNT100;
   1:  PR[GP1:91,1] = PR[GP1:90,1] + -63.473;
   1:  PR[GP1:91,2] = PR[GP1:90,2] + 19.272;
   1:L PR[91] R[100]mm/sec CNT100;
   1:  PR[GP1:91,1] = PR[GP1:90,1] + -67.620;
   1:  PR[GP1:91,2] = PR[GP1:90,2] + 10.996;
   1:L PR[91] R[100]mm/sec CNT100;
   1:  PR[GP1:91,1] = PR[GP1:90,1] + -68.186;
   1:  PR[GP1:91,2] = PR[GP1:90,2] + 9.075;
   1:L PR[91] R[100]mm/sec CNT100;
   1:  PR[GP1:91,1] = PR[GP1:90,1] + -69.339;
   1:  PR[GP1:91,2] = PR[GP1:90,2] + 1.676;
   1:L PR[91] R[100]mm/sec CNT100;
   1:  PR[GP1:91,1] = PR[GP1:90,1] + -69.495;
   1:  PR[GP1:91,2] = PR[GP1:90,2] + -0.052;
   1:L PR[91] R[100]mm/sec CNT100;
   1:  PR[GP1:91,1] = PR[GP1:90,1] + -68.354;
   1:  PR[GP1:91,2] = PR[GP1:90,2] + -7.274;
   1:L PR[91] R[100]mm/sec CNT100;
   1:  PR[GP1:91,1] = PR[GP1:90,1] + -68.180;
   1:  PR[GP1:91,2] = PR[GP1:90,2] + -9.238;
   1:L PR[91] R[100]mm/sec CNT100;
   1:  PR[GP1:91,1] = PR[GP1:90,1] + -67.620;
   1:  PR[GP1:91,2] = PR[GP1:90,2] + -11.140;
   1:L PR[91] R[100]mm/sec CNT100;
   1:  PR[GP1:91,1] = PR[GP1:90,1] + -63.473;
   1:  PR[GP1:91,2] = PR[GP1:90,2] + -19.416;
   1:L PR[91] R[100]mm/sec CNT100;
   1:  PR[GP1:91,1] = PR[GP1:90,1] + -61.728;
   1:  PR[GP1:91,2] = PR[GP1:90,2] + -21.680;
   1:L PR[91] R[100]mm/sec CNT100;
   1:  PR[GP1:91,1] = PR[GP1:90,1] + -57.902;
   1:  PR[GP1:91,2] = PR[GP1:90,2] + -25.702;
   1:L PR[91] R[100]mm/sec CNT100;
   1:  PR[GP1:91,1] = PR[GP1:90,1] + -55.328;
   1:  PR[GP1:91,2] = PR[GP1:90,2] + -28.010;
   1:L PR[91] R[100]mm/sec CNT100;
   1:  PR[GP1:91,1] = PR[GP1:90,1] + -51.920;
   1:  PR[GP1:91,2] = PR[GP1:90,2] + -29.927;
   1:L PR[91] R[100]mm/sec CNT100;
   1:  PR[GP1:91,1] = PR[GP1:90,1] + -48.463;
   1:  PR[GP1:91,2] = PR[GP1:90,2] + -32.117;
   1:L PR[91] R[100]mm/sec CNT100;
   1:  PR[GP1:91,1] = PR[GP1:90,1] + -43.433;
   1:  PR[GP1:91,2] = PR[GP1:90,2] + -34.097;
   1:L PR[91] R[100]mm/sec CNT100;
   1:  PR[GP1:91,1] = PR[GP1:90,1] + -42.221;
   1:  PR[GP1:91,2] = PR[GP1:90,2] + -34.382;
   1:L PR[91] R[100]mm/sec CNT100;
   1:  PR[GP1:91,1] = PR[GP1:90,1] + -36.365;
   1:  PR[GP1:91,2] = PR[GP1:90,2] + -35.626;
   1:L PR[91] R[100]mm/sec CNT100;
   1:  PR[GP1:91,1] = PR[GP1:90,1] + -30.042;
   1:  PR[GP1:91,2] = PR[GP1:90,2] + -35.870;
   1:L PR[91] R[100]mm/sec CNT100;
   1:  PR[GP1:91,1] = PR[GP1:90,1] + -28.975;
   1:  PR[GP1:91,2] = PR[GP1:90,2] + -35.873;
   1:L PR[91] R[100]mm/sec CNT100;
   1:  PR[GP1:91,1] = PR[GP1:90,1] + -22.795;
   1:  PR[GP1:91,2] = PR[GP1:90,2] + -35.066;
   1:L PR[91] R[100]mm/sec CNT100;
   1:  PR[GP1:91,1] = PR[GP1:90,1] + -17.514;
   1:  PR[GP1:91,2] = PR[GP1:90,2] + -33.385;
   1:L PR[91] R[100]mm/sec CNT100;
   1:  PR[GP1:91,1] = PR[GP1:90,1] + -15.062;
   1:  PR[GP1:91,2] = PR[GP1:90,2] + -32.533;
   1:L PR[91] R[100]mm/sec CNT100;
   1:  PR[GP1:91,1] = PR[GP1:90,1] + -10.289;
   1:  PR[GP1:91,2] = PR[GP1:90,2] + -30.036;
   1:L PR[91] R[100]mm/sec CNT100;
   1:  PR[GP1:91,1] = PR[GP1:90,1] + -8.438;
   1:  PR[GP1:91,2] = PR[GP1:90,2] + -28.691;
   1:L PR[91] R[100]mm/sec CNT100;
   1:  PR[GP1:91,1] = PR[GP1:90,1] + -5.667;
   1:  PR[GP1:91,2] = PR[GP1:90,2] + -26.521;
   1:L PR[91] R[100]mm/sec CNT100;
   1:  PR[GP1:91,1] = PR[GP1:90,1] + -3.550;
   1:  PR[GP1:91,2] = PR[GP1:90,2] + -24.065;
   1:L PR[91] R[100]mm/sec CNT100;
   1:  PR[GP1:91,1] = PR[GP1:90,1] + -1.300;
   1:  PR[GP1:91,2] = PR[GP1:90,2] + -23.582;
   1:L PR[91] R[100]mm/sec CNT100;
   1:  PR[GP1:91,1] = PR[GP1:90,1] + 0.681;
   1:  PR[GP1:91,2] = PR[GP1:90,2] + -22.532;
   1:L PR[91] R[100]mm/sec CNT100;
   1:  PR[GP1:91,1] = PR[GP1:90,1] + 3.822;
   1:  PR[GP1:91,2] = PR[GP1:90,2] + -24.128;
   1:L PR[91] R[100]mm/sec CNT100;
   1:  PR[GP1:91,1] = PR[GP1:90,1] + 5.904;
   1:  PR[GP1:91,2] = PR[GP1:90,2] + -26.546;
   1:L PR[91] R[100]mm/sec CNT100;
   1:  PR[GP1:91,1] = PR[GP1:90,1] + 8.662;
   1:  PR[GP1:91,2] = PR[GP1:90,2] + -28.704;
   1:L PR[91] R[100]mm/sec CNT100;
   1:  PR[GP1:91,1] = PR[GP1:90,1] + 10.517;
   1:  PR[GP1:91,2] = PR[GP1:90,2] + -30.051;
   1:L PR[91] R[100]mm/sec CNT100;
   1:  PR[GP1:91,1] = PR[GP1:90,1] + 15.254;
   1:  PR[GP1:91,2] = PR[GP1:90,2] + -32.523;
   1:L PR[91] R[100]mm/sec CNT100;
   1:  PR[GP1:91,1] = PR[GP1:90,1] + 21.107;
   1:  PR[GP1:91,2] = PR[GP1:90,2] + -34.404;
   1:L PR[91] R[100]mm/sec CNT100;
   1:  PR[GP1:91,1] = PR[GP1:90,1] + 23.011;
   1:  PR[GP1:91,2] = PR[GP1:90,2] + -35.063;
   1:L PR[91] R[100]mm/sec CNT100;
   1:  PR[GP1:91,1] = PR[GP1:90,1] + 29.165;
   1:  PR[GP1:91,2] = PR[GP1:90,2] + -35.872;
   1:L PR[91] R[100]mm/sec CNT100;
   1:  PR[GP1:91,1] = PR[GP1:90,1] + 36.536;
   1:  PR[GP1:91,2] = PR[GP1:90,2] + -35.632;
   1:L PR[91] R[100]mm/sec CNT100;
   1:  PR[GP1:91,1] = PR[GP1:90,1] + 43.606;
   1:  PR[GP1:91,2] = PR[GP1:90,2] + -34.105;
   1:L PR[91] R[100]mm/sec CNT100;
   1:  PR[GP1:91,1] = PR[GP1:90,1] + 48.666;
   1:  PR[GP1:91,2] = PR[GP1:90,2] + -32.124;
   1:L PR[91] R[100]mm/sec CNT100;
   1:  PR[GP1:91,1] = PR[GP1:90,1] + 51.527;
   1:  PR[GP1:91,2] = PR[GP1:90,2] + -30.499;
   1:L PR[91] R[100]mm/sec CNT100;
   1:  PR[GP1:91,1] = PR[GP1:90,1] + 55.494;
   1:  PR[GP1:91,2] = PR[GP1:90,2] + -28.053;
   1:L PR[91] R[100]mm/sec CNT100;
   1:  PR[GP1:91,1] = PR[GP1:90,1] + 58.075;
   1:  PR[GP1:91,2] = PR[GP1:90,2] + -25.746;
   1:L PR[91] R[100]mm/sec CNT100;
   1:  PR[GP1:91,1] = PR[GP1:90,1] + 61.899;
   1:  PR[GP1:91,2] = PR[GP1:90,2] + -21.713;
   1:L PR[91] R[100]mm/sec CNT100;
   1:  PR[GP1:91,1] = PR[GP1:90,1] + 63.670;
   1:  PR[GP1:91,2] = PR[GP1:90,2] + -19.421;
   1:L PR[91] R[100]mm/sec CNT100;
   1:  PR[GP1:91,1] = PR[GP1:90,1] + 66.714;
   1:  PR[GP1:91,2] = PR[GP1:90,2] + -13.364;
   1:L PR[91] R[100]mm/sec CNT100;
   1:  PR[GP1:91,1] = PR[GP1:90,1] + 67.825;
   1:  PR[GP1:91,2] = PR[GP1:90,2] + -11.187;
   1:L PR[91] R[100]mm/sec CNT100;
   1:  PR[GP1:91,1] = PR[GP1:90,1] + 68.390;
   1:  PR[GP1:91,2] = PR[GP1:90,2] + -9.293;
   1:L PR[91] R[100]mm/sec CNT100;
   1:  PR[GP1:91,1] = PR[GP1:90,1] + 69.544;
   1:  PR[GP1:91,2] = PR[GP1:90,2] + -1.871;
   1:L PR[91] R[100]mm/sec CNT100;
   1:  PR[GP1:91,1] = PR[GP1:90,1] + 69.708;
   1:  PR[GP1:91,2] = PR[GP1:90,2] + -0.092;
   1:L PR[91] R[100]mm/sec CNT100;
   1:  PR[GP1:91,1] = PR[GP1:90,1] + 68.567;
   1:  PR[GP1:91,2] = PR[GP1:90,2] + 7.150;
   1:L PR[91] R[100]mm/sec CNT100;
   1:  PR[GP1:91,1] = PR[GP1:90,1] + 68.385;
   1:  PR[GP1:91,2] = PR[GP1:90,2] + 9.168;
   1:L PR[91] R[100]mm/sec CNT100;
   1:  PR[GP1:91,1] = PR[GP1:90,1] + 67.824;
   1:  PR[GP1:91,2] = PR[GP1:90,2] + 11.045;
   1:L PR[91] R[100]mm/sec CNT100;
   1:  PR[GP1:91,1] = PR[GP1:90,1] + 64.820;
   1:  PR[GP1:91,2] = PR[GP1:90,2] + 17.028;
   1:L PR[91] R[100]mm/sec CNT100;
   1:  PR[GP1:91,1] = PR[GP1:90,1] + 63.672;
   1:  PR[GP1:91,2] = PR[GP1:90,2] + 19.276;
   1:L PR[91] R[100]mm/sec CNT100;
   1:  PR[GP1:91,1] = PR[GP1:90,1] + 61.899;
   1:  PR[GP1:91,2] = PR[GP1:90,2] + 21.569;
   1:L PR[91] R[100]mm/sec CNT100;
   1:  PR[GP1:91,1] = PR[GP1:90,1] + 58.075;
   1:  PR[GP1:91,2] = PR[GP1:90,2] + 25.602;
   1:L PR[91] R[100]mm/sec CNT100;
   1:  PR[GP1:91,1] = PR[GP1:90,1] + 55.503;
   1:  PR[GP1:91,2] = PR[GP1:90,2] + 27.901;
   1:L PR[91] R[100]mm/sec CNT100;
   1:  PR[GP1:91,1] = PR[GP1:90,1] + 52.099;
   1:  PR[GP1:91,2] = PR[GP1:90,2] + 29.813;
   1:L PR[91] R[100]mm/sec CNT100;
   1:  PR[GP1:91,1] = PR[GP1:90,1] + 48.653;
   1:  PR[GP1:91,2] = PR[GP1:90,2] + 31.985;
   1:L PR[91] R[100]mm/sec CNT100;
   1:  PR[GP1:91,1] = PR[GP1:90,1] + 43.600;
   1:  PR[GP1:91,2] = PR[GP1:90,2] + 33.963;
   1:L PR[91] R[100]mm/sec CNT100;
   1:  PR[GP1:91,1] = PR[GP1:90,1] + 42.398;
   1:  PR[GP1:91,2] = PR[GP1:90,2] + 34.247;
   1:L PR[91] R[100]mm/sec CNT100;
   1:  PR[GP1:91,1] = PR[GP1:90,1] + 36.536;
   1:  PR[GP1:91,2] = PR[GP1:90,2] + 35.488;
   1:L PR[91] R[100]mm/sec CNT100;
   1:  PR[GP1:91,1] = PR[GP1:90,1] + 30.244;
   1:  PR[GP1:91,2] = PR[GP1:90,2] + 35.726;
   1:L PR[91] R[100]mm/sec CNT100;
   1:  PR[GP1:91,1] = PR[GP1:90,1] + 29.175;
   1:  PR[GP1:91,2] = PR[GP1:90,2] + 35.729;
   1:L PR[91] R[100]mm/sec CNT100;
   1:  PR[GP1:91,1] = PR[GP1:90,1] + 23.006;
   1:  PR[GP1:91,2] = PR[GP1:90,2] + 34.918;
   1:L PR[91] R[100]mm/sec CNT100;
   1:  PR[GP1:91,1] = PR[GP1:90,1] + 17.719;
   1:  PR[GP1:91,2] = PR[GP1:90,2] + 33.236;
   1:L PR[91] R[100]mm/sec CNT100;
   1:  PR[GP1:91,1] = PR[GP1:90,1] + 15.265;
   1:  PR[GP1:91,2] = PR[GP1:90,2] + 32.385;
   1:L PR[91] R[100]mm/sec CNT100;
   1:  PR[GP1:91,1] = PR[GP1:90,1] + 10.516;
   1:  PR[GP1:91,2] = PR[GP1:90,2] + 29.907;
   1:L PR[91] R[100]mm/sec CNT100;
   1:  PR[GP1:91,1] = PR[GP1:90,1] + 9.178;
   1:  PR[GP1:91,2] = PR[GP1:90,2] + 28.962;
   1:L PR[91] R[100]mm/sec CNT100;
   1:  PR[GP1:91,1] = PR[GP1:90,1] + 6.147;
   1:  PR[GP1:91,2] = PR[GP1:90,2] + 26.590;
   1:L PR[91] R[100]mm/sec CNT100;
   1:  PR[GP1:91,1] = PR[GP1:90,1] + 3.805;
   1:  PR[GP1:91,2] = PR[GP1:90,2] + 23.864;
   1:L PR[91] R[100]mm/sec CNT100;
   1:  PR[GP1:91,1] = PR[GP1:90,1] + 2.779;
   1:  PR[GP1:91,2] = PR[GP1:90,2] + 23.459;
   1:L PR[91] R[100]mm/sec CNT100;
   1:  PR[GP1:91,1] = PR[GP1:90,1] + 0.795;
   1:  PR[GP1:91,2] = PR[GP1:90,2] + 22.445;
   1:L PR[91] R[100]mm/sec CNT100;
   1:  ! -- Layer/Ebene 77 -- !;
   1:  PR[91] = PR[90];
   1:  PR[GP1:91,1] = PR[GP1:90,1] + -1.389;
   1:  PR[GP1:91,2] = PR[GP1:90,2] + 23.061;
   1:  PR[GP1:91,3] = PR[GP1:90,3] + 47.275;
   1:L PR[91] R[100]mm/sec CNT100;
   1:  PR[GP1:91,1] = PR[GP1:90,1] + -3.577;
   1:  PR[GP1:91,2] = PR[GP1:90,2] + 24.174;
   1:L PR[91] R[100]mm/sec CNT100;
   1:  PR[GP1:91,1] = PR[GP1:90,1] + -5.751;
   1:  PR[GP1:91,2] = PR[GP1:90,2] + 26.702;
   1:L PR[91] R[100]mm/sec CNT100;
   1:  PR[GP1:91,1] = PR[GP1:90,1] + -8.624;
   1:  PR[GP1:91,2] = PR[GP1:90,2] + 28.952;
   1:L PR[91] R[100]mm/sec CNT100;
   1:  PR[GP1:91,1] = PR[GP1:90,1] + -10.078;
   1:  PR[GP1:91,2] = PR[GP1:90,2] + 29.979;
   1:L PR[91] R[100]mm/sec CNT100;
   1:  PR[GP1:91,1] = PR[GP1:90,1] + -14.718;
   1:  PR[GP1:91,2] = PR[GP1:90,2] + 32.407;
   1:L PR[91] R[100]mm/sec CNT100;
   1:  PR[GP1:91,1] = PR[GP1:90,1] + -20.404;
   1:  PR[GP1:91,2] = PR[GP1:90,2] + 34.234;
   1:L PR[91] R[100]mm/sec CNT100;
   1:  PR[GP1:91,1] = PR[GP1:90,1] + -22.607;
   1:  PR[GP1:91,2] = PR[GP1:90,2] + 34.995;
   1:L PR[91] R[100]mm/sec CNT100;
   1:  PR[GP1:91,1] = PR[GP1:90,1] + -28.616;
   1:  PR[GP1:91,2] = PR[GP1:90,2] + 35.780;
   1:L PR[91] R[100]mm/sec CNT100;
   1:  PR[GP1:91,1] = PR[GP1:90,1] + -35.627;
   1:  PR[GP1:91,2] = PR[GP1:90,2] + 35.539;
   1:L PR[91] R[100]mm/sec CNT100;
   1:  PR[GP1:91,1] = PR[GP1:90,1] + -36.186;
   1:  PR[GP1:91,2] = PR[GP1:90,2] + 35.537;
   1:L PR[91] R[100]mm/sec CNT100;
   1:  PR[GP1:91,1] = PR[GP1:90,1] + -43.043;
   1:  PR[GP1:91,2] = PR[GP1:90,2] + 34.055;
   1:L PR[91] R[100]mm/sec CNT100;
   1:  PR[GP1:91,1] = PR[GP1:90,1] + -48.480;
   1:  PR[GP1:91,2] = PR[GP1:90,2] + 31.915;
   1:L PR[91] R[100]mm/sec CNT100;
   1:  PR[GP1:91,1] = PR[GP1:90,1] + -50.718;
   1:  PR[GP1:91,2] = PR[GP1:90,2] + 30.642;
   1:L PR[91] R[100]mm/sec CNT100;
   1:  PR[GP1:91,1] = PR[GP1:90,1] + -55.106;
   1:  PR[GP1:91,2] = PR[GP1:90,2] + 27.924;
   1:L PR[91] R[100]mm/sec CNT100;
   1:  PR[GP1:91,1] = PR[GP1:90,1] + -57.958;
   1:  PR[GP1:91,2] = PR[GP1:90,2] + 25.367;
   1:L PR[91] R[100]mm/sec CNT100;
   1:  PR[GP1:91,1] = PR[GP1:90,1] + -61.361;
   1:  PR[GP1:91,2] = PR[GP1:90,2] + 21.789;
   1:L PR[91] R[100]mm/sec CNT100;
   1:  PR[GP1:91,1] = PR[GP1:90,1] + -63.348;
   1:  PR[GP1:91,2] = PR[GP1:90,2] + 19.211;
   1:L PR[91] R[100]mm/sec CNT100;
   1:  PR[GP1:91,1] = PR[GP1:90,1] + -67.403;
   1:  PR[GP1:91,2] = PR[GP1:90,2] + 11.122;
   1:L PR[91] R[100]mm/sec CNT100;
   1:  PR[GP1:91,1] = PR[GP1:90,1] + -68.069;
   1:  PR[GP1:91,2] = PR[GP1:90,2] + 8.861;
   1:L PR[91] R[100]mm/sec CNT100;
   1:  PR[GP1:91,1] = PR[GP1:90,1] + -69.133;
   1:  PR[GP1:91,2] = PR[GP1:90,2] + 2.039;
   1:L PR[91] R[100]mm/sec CNT100;
   1:  PR[GP1:91,1] = PR[GP1:90,1] + -69.321;
   1:  PR[GP1:91,2] = PR[GP1:90,2] + -0.052;
   1:L PR[91] R[100]mm/sec CNT100;
   1:  PR[GP1:91,1] = PR[GP1:90,1] + -68.267;
   1:  PR[GP1:91,2] = PR[GP1:90,2] + -6.721;
   1:L PR[91] R[100]mm/sec CNT100;
   1:  PR[GP1:91,1] = PR[GP1:90,1] + -68.064;
   1:  PR[GP1:91,2] = PR[GP1:90,2] + -9.024;
   1:L PR[91] R[100]mm/sec CNT100;
   1:  PR[GP1:91,1] = PR[GP1:90,1] + -67.403;
   1:  PR[GP1:91,2] = PR[GP1:90,2] + -11.266;
   1:L PR[91] R[100]mm/sec CNT100;
   1:  PR[GP1:91,1] = PR[GP1:90,1] + -63.348;
   1:  PR[GP1:91,2] = PR[GP1:90,2] + -19.355;
   1:L PR[91] R[100]mm/sec CNT100;
   1:  PR[GP1:91,1] = PR[GP1:90,1] + -61.361;
   1:  PR[GP1:91,2] = PR[GP1:90,2] + -21.933;
   1:L PR[91] R[100]mm/sec CNT100;
   1:  PR[GP1:91,1] = PR[GP1:90,1] + -57.958;
   1:  PR[GP1:91,2] = PR[GP1:90,2] + -25.511;
   1:L PR[91] R[100]mm/sec CNT100;
   1:  PR[GP1:91,1] = PR[GP1:90,1] + -55.115;
   1:  PR[GP1:91,2] = PR[GP1:90,2] + -28.059;
   1:L PR[91] R[100]mm/sec CNT100;
   1:  PR[GP1:91,1] = PR[GP1:90,1] + -52.196;
   1:  PR[GP1:91,2] = PR[GP1:90,2] + -29.702;
   1:L PR[91] R[100]mm/sec CNT100;
   1:  PR[GP1:91,1] = PR[GP1:90,1] + -48.467;
   1:  PR[GP1:91,2] = PR[GP1:90,2] + -32.064;
   1:L PR[91] R[100]mm/sec CNT100;
   1:  PR[GP1:91,1] = PR[GP1:90,1] + -43.038;
   1:  PR[GP1:91,2] = PR[GP1:90,2] + -34.201;
   1:L PR[91] R[100]mm/sec CNT100;
   1:  PR[GP1:91,1] = PR[GP1:90,1] + -42.460;
   1:  PR[GP1:91,2] = PR[GP1:90,2] + -34.337;
   1:L PR[91] R[100]mm/sec CNT100;
   1:  PR[GP1:91,1] = PR[GP1:90,1] + -36.176;
   1:  PR[GP1:91,2] = PR[GP1:90,2] + -35.683;
   1:L PR[91] R[100]mm/sec CNT100;
   1:  PR[GP1:91,1] = PR[GP1:90,1] + -29.996;
   1:  PR[GP1:91,2] = PR[GP1:90,2] + -35.921;
   1:L PR[91] R[100]mm/sec CNT100;
   1:  PR[GP1:91,1] = PR[GP1:90,1] + -28.623;
   1:  PR[GP1:91,2] = PR[GP1:90,2] + -35.925;
   1:L PR[91] R[100]mm/sec CNT100;
   1:  PR[GP1:91,1] = PR[GP1:90,1] + -22.596;
   1:  PR[GP1:91,2] = PR[GP1:90,2] + -35.138;
   1:L PR[91] R[100]mm/sec CNT100;
   1:  PR[GP1:91,1] = PR[GP1:90,1] + -17.446;
   1:  PR[GP1:91,2] = PR[GP1:90,2] + -33.499;
   1:L PR[91] R[100]mm/sec CNT100;
   1:  PR[GP1:91,1] = PR[GP1:90,1] + -14.720;
   1:  PR[GP1:91,2] = PR[GP1:90,2] + -32.551;
   1:L PR[91] R[100]mm/sec CNT100;
   1:  PR[GP1:91,1] = PR[GP1:90,1] + -10.078;
   1:  PR[GP1:91,2] = PR[GP1:90,2] + -30.123;
   1:L PR[91] R[100]mm/sec CNT100;
   1:  PR[GP1:91,1] = PR[GP1:90,1] + -8.064;
   1:  PR[GP1:91,2] = PR[GP1:90,2] + -28.660;
   1:L PR[91] R[100]mm/sec CNT100;
   1:  PR[GP1:91,1] = PR[GP1:90,1] + -5.494;
   1:  PR[GP1:91,2] = PR[GP1:90,2] + -26.647;
   1:L PR[91] R[100]mm/sec CNT100;
   1:  PR[GP1:91,1] = PR[GP1:90,1] + -3.520;
   1:  PR[GP1:91,2] = PR[GP1:90,2] + -24.358;
   1:L PR[91] R[100]mm/sec CNT100;
   1:  PR[GP1:91,1] = PR[GP1:90,1] + -1.133;
   1:  PR[GP1:91,2] = PR[GP1:90,2] + -23.846;
   1:L PR[91] R[100]mm/sec CNT100;
   1:  PR[GP1:91,1] = PR[GP1:90,1] + 0.723;
   1:  PR[GP1:91,2] = PR[GP1:90,2] + -22.862;
   1:L PR[91] R[100]mm/sec CNT100;
   1:  PR[GP1:91,1] = PR[GP1:90,1] + 3.792;
   1:  PR[GP1:91,2] = PR[GP1:90,2] + -24.421;
   1:L PR[91] R[100]mm/sec CNT100;
   1:  PR[GP1:91,1] = PR[GP1:90,1] + 5.729;
   1:  PR[GP1:91,2] = PR[GP1:90,2] + -26.670;
   1:L PR[91] R[100]mm/sec CNT100;
   1:  PR[GP1:91,1] = PR[GP1:90,1] + 8.287;
   1:  PR[GP1:91,2] = PR[GP1:90,2] + -28.672;
   1:L PR[91] R[100]mm/sec CNT100;
   1:  PR[GP1:91,1] = PR[GP1:90,1] + 10.305;
   1:  PR[GP1:91,2] = PR[GP1:90,2] + -30.138;
   1:L PR[91] R[100]mm/sec CNT100;
   1:  PR[GP1:91,1] = PR[GP1:90,1] + 14.912;
   1:  PR[GP1:91,2] = PR[GP1:90,2] + -32.542;
   1:L PR[91] R[100]mm/sec CNT100;
   1:  PR[GP1:91,1] = PR[GP1:90,1] + 20.606;
   1:  PR[GP1:91,2] = PR[GP1:90,2] + -34.371;
   1:L PR[91] R[100]mm/sec CNT100;
   1:  PR[GP1:91,1] = PR[GP1:90,1] + 22.812;
   1:  PR[GP1:91,2] = PR[GP1:90,2] + -35.135;
   1:L PR[91] R[100]mm/sec CNT100;
   1:  PR[GP1:91,1] = PR[GP1:90,1] + 28.813;
   1:  PR[GP1:91,2] = PR[GP1:90,2] + -35.924;
   1:L PR[91] R[100]mm/sec CNT100;
   1:  PR[GP1:91,1] = PR[GP1:90,1] + 35.791;
   1:  PR[GP1:91,2] = PR[GP1:90,2] + -35.689;
   1:L PR[91] R[100]mm/sec CNT100;
   1:  PR[GP1:91,1] = PR[GP1:90,1] + 36.357;
   1:  PR[GP1:91,2] = PR[GP1:90,2] + -35.687;
   1:L PR[91] R[100]mm/sec CNT100;
   1:  PR[GP1:91,1] = PR[GP1:90,1] + 43.208;
   1:  PR[GP1:91,2] = PR[GP1:90,2] + -34.210;
   1:L PR[91] R[100]mm/sec CNT100;
   1:  PR[GP1:91,1] = PR[GP1:90,1] + 48.668;
   1:  PR[GP1:91,2] = PR[GP1:90,2] + -32.072;
   1:L PR[91] R[100]mm/sec CNT100;
   1:  PR[GP1:91,1] = PR[GP1:90,1] + 50.900;
   1:  PR[GP1:91,2] = PR[GP1:90,2] + -30.804;
   1:L PR[91] R[100]mm/sec CNT100;
   1:  PR[GP1:91,1] = PR[GP1:90,1] + 55.277;
   1:  PR[GP1:91,2] = PR[GP1:90,2] + -28.106;
   1:L PR[91] R[100]mm/sec CNT100;
   1:  PR[GP1:91,1] = PR[GP1:90,1] + 58.127;
   1:  PR[GP1:91,2] = PR[GP1:90,2] + -25.559;
   1:L PR[91] R[100]mm/sec CNT100;
   1:  PR[GP1:91,1] = PR[GP1:90,1] + 61.527;
   1:  PR[GP1:91,2] = PR[GP1:90,2] + -21.973;
   1:L PR[91] R[100]mm/sec CNT100;
   1:  PR[GP1:91,1] = PR[GP1:90,1] + 63.543;
   1:  PR[GP1:91,2] = PR[GP1:90,2] + -19.363;
   1:L PR[91] R[100]mm/sec CNT100;
   1:  PR[GP1:91,1] = PR[GP1:90,1] + 66.304;
   1:  PR[GP1:91,2] = PR[GP1:90,2] + -13.870;
   1:L PR[91] R[100]mm/sec CNT100;
   1:  PR[GP1:91,1] = PR[GP1:90,1] + 67.607;
   1:  PR[GP1:91,2] = PR[GP1:90,2] + -11.317;
   1:L PR[91] R[100]mm/sec CNT100;
   1:  PR[GP1:91,1] = PR[GP1:90,1] + 68.272;
   1:  PR[GP1:91,2] = PR[GP1:90,2] + -9.087;
   1:L PR[91] R[100]mm/sec CNT100;
   1:  PR[GP1:91,1] = PR[GP1:90,1] + 69.336;
   1:  PR[GP1:91,2] = PR[GP1:90,2] + -2.245;
   1:L PR[91] R[100]mm/sec CNT100;
   1:  PR[GP1:91,1] = PR[GP1:90,1] + 69.534;
   1:  PR[GP1:91,2] = PR[GP1:90,2] + -0.092;
   1:L PR[91] R[100]mm/sec CNT100;
   1:  PR[GP1:91,1] = PR[GP1:90,1] + 68.480;
   1:  PR[GP1:91,2] = PR[GP1:90,2] + 6.595;
   1:L PR[91] R[100]mm/sec CNT100;
   1:  PR[GP1:91,1] = PR[GP1:90,1] + 68.266;
   1:  PR[GP1:91,2] = PR[GP1:90,2] + 8.962;
   1:L PR[91] R[100]mm/sec CNT100;
   1:  PR[GP1:91,1] = PR[GP1:90,1] + 67.606;
   1:  PR[GP1:91,2] = PR[GP1:90,2] + 11.175;
   1:L PR[91] R[100]mm/sec CNT100;
   1:  PR[GP1:91,1] = PR[GP1:90,1] + 64.852;
   1:  PR[GP1:91,2] = PR[GP1:90,2] + 16.661;
   1:L PR[91] R[100]mm/sec CNT100;
   1:  PR[GP1:91,1] = PR[GP1:90,1] + 63.545;
   1:  PR[GP1:91,2] = PR[GP1:90,2] + 19.218;
   1:L PR[91] R[100]mm/sec CNT100;
   1:  PR[GP1:91,1] = PR[GP1:90,1] + 61.527;
   1:  PR[GP1:91,2] = PR[GP1:90,2] + 21.829;
   1:L PR[91] R[100]mm/sec CNT100;
   1:  PR[GP1:91,1] = PR[GP1:90,1] + 58.127;
   1:  PR[GP1:91,2] = PR[GP1:90,2] + 25.415;
   1:L PR[91] R[100]mm/sec CNT100;
   1:  PR[GP1:91,1] = PR[GP1:90,1] + 55.286;
   1:  PR[GP1:91,2] = PR[GP1:90,2] + 27.954;
   1:L PR[91] R[100]mm/sec CNT100;
   1:  PR[GP1:91,1] = PR[GP1:90,1] + 52.373;
   1:  PR[GP1:91,2] = PR[GP1:90,2] + 29.591;
   1:L PR[91] R[100]mm/sec CNT100;
   1:  PR[GP1:91,1] = PR[GP1:90,1] + 48.656;
   1:  PR[GP1:91,2] = PR[GP1:90,2] + 31.933;
   1:L PR[91] R[100]mm/sec CNT100;
   1:  PR[GP1:91,1] = PR[GP1:90,1] + 43.202;
   1:  PR[GP1:91,2] = PR[GP1:90,2] + 34.068;
   1:L PR[91] R[100]mm/sec CNT100;
   1:  PR[GP1:91,1] = PR[GP1:90,1] + 42.635;
   1:  PR[GP1:91,2] = PR[GP1:90,2] + 34.202;
   1:L PR[91] R[100]mm/sec CNT100;
   1:  PR[GP1:91,1] = PR[GP1:90,1] + 36.348;
   1:  PR[GP1:91,2] = PR[GP1:90,2] + 35.545;
   1:L PR[91] R[100]mm/sec CNT100;
   1:  PR[GP1:91,1] = PR[GP1:90,1] + 30.199;
   1:  PR[GP1:91,2] = PR[GP1:90,2] + 35.777;
   1:L PR[91] R[100]mm/sec CNT100;
   1:  PR[GP1:91,1] = PR[GP1:90,1] + 28.824;
   1:  PR[GP1:91,2] = PR[GP1:90,2] + 35.782;
   1:L PR[91] R[100]mm/sec CNT100;
   1:  PR[GP1:91,1] = PR[GP1:90,1] + 22.808;
   1:  PR[GP1:91,2] = PR[GP1:90,2] + 34.991;
   1:L PR[91] R[100]mm/sec CNT100;
   1:  PR[GP1:91,1] = PR[GP1:90,1] + 17.651;
   1:  PR[GP1:91,2] = PR[GP1:90,2] + 33.350;
   1:L PR[91] R[100]mm/sec CNT100;
   1:  PR[GP1:91,1] = PR[GP1:90,1] + 14.923;
   1:  PR[GP1:91,2] = PR[GP1:90,2] + 32.404;
   1:L PR[91] R[100]mm/sec CNT100;
   1:  PR[GP1:91,1] = PR[GP1:90,1] + 10.305;
   1:  PR[GP1:91,2] = PR[GP1:90,2] + 29.994;
   1:L PR[91] R[100]mm/sec CNT100;
   1:  PR[GP1:91,1] = PR[GP1:90,1] + 8.848;
   1:  PR[GP1:91,2] = PR[GP1:90,2] + 28.965;
   1:L PR[91] R[100]mm/sec CNT100;
   1:  PR[GP1:91,1] = PR[GP1:90,1] + 5.989;
   1:  PR[GP1:91,2] = PR[GP1:90,2] + 26.728;
   1:L PR[91] R[100]mm/sec CNT100;
   1:  PR[GP1:91,1] = PR[GP1:90,1] + 3.775;
   1:  PR[GP1:91,2] = PR[GP1:90,2] + 24.151;
   1:L PR[91] R[100]mm/sec CNT100;
   1:  PR[GP1:91,1] = PR[GP1:90,1] + 2.690;
   1:  PR[GP1:91,2] = PR[GP1:90,2] + 23.723;
   1:L PR[91] R[100]mm/sec CNT100;
   1:  PR[GP1:91,1] = PR[GP1:90,1] + 0.836;
   1:  PR[GP1:91,2] = PR[GP1:90,2] + 22.775;
   1:L PR[91] R[100]mm/sec CNT100;
   1:  ! -- Layer/Ebene 78 -- !;
   1:  PR[91] = PR[90];
   1:  PR[GP1:91,1] = PR[GP1:90,1] + -1.478;
   1:  PR[GP1:91,2] = PR[GP1:90,2] + 23.407;
   1:  PR[GP1:91,3] = PR[GP1:90,3] + 47.885;
   1:L PR[91] R[100]mm/sec CNT100;
   1:  PR[GP1:91,1] = PR[GP1:90,1] + -3.547;
   1:  PR[GP1:91,2] = PR[GP1:90,2] + 24.460;
   1:L PR[91] R[100]mm/sec CNT100;
   1:  PR[GP1:91,1] = PR[GP1:90,1] + -5.596;
   1:  PR[GP1:91,2] = PR[GP1:90,2] + 26.842;
   1:L PR[91] R[100]mm/sec CNT100;
   1:  PR[GP1:91,1] = PR[GP1:90,1] + -8.294;
   1:  PR[GP1:91,2] = PR[GP1:90,2] + 28.955;
   1:L PR[91] R[100]mm/sec CNT100;
   1:  PR[GP1:91,1] = PR[GP1:90,1] + -9.867;
   1:  PR[GP1:91,2] = PR[GP1:90,2] + 30.066;
   1:L PR[91] R[100]mm/sec CNT100;
   1:  PR[GP1:91,1] = PR[GP1:90,1] + -14.376;
   1:  PR[GP1:91,2] = PR[GP1:90,2] + 32.426;
   1:L PR[91] R[100]mm/sec CNT100;
   1:  PR[GP1:91,1] = PR[GP1:90,1] + -19.903;
   1:  PR[GP1:91,2] = PR[GP1:90,2] + 34.201;
   1:L PR[91] R[100]mm/sec CNT100;
   1:  PR[GP1:91,1] = PR[GP1:90,1] + -22.409;
   1:  PR[GP1:91,2] = PR[GP1:90,2] + 35.067;
   1:L PR[91] R[100]mm/sec CNT100;
   1:  PR[GP1:91,1] = PR[GP1:90,1] + -28.264;
   1:  PR[GP1:91,2] = PR[GP1:90,2] + 35.833;
   1:L PR[91] R[100]mm/sec CNT100;
   1:  PR[GP1:91,1] = PR[GP1:90,1] + -35.098;
   1:  PR[GP1:91,2] = PR[GP1:90,2] + 35.598;
   1:L PR[91] R[100]mm/sec CNT100;
   1:  PR[GP1:91,1] = PR[GP1:90,1] + -35.998;
   1:  PR[GP1:91,2] = PR[GP1:90,2] + 35.593;
   1:L PR[91] R[100]mm/sec CNT100;
   1:  PR[GP1:91,1] = PR[GP1:90,1] + -42.650;
   1:  PR[GP1:91,2] = PR[GP1:90,2] + 34.158;
   1:L PR[91] R[100]mm/sec CNT100;
   1:  PR[GP1:91,1] = PR[GP1:90,1] + -48.485;
   1:  PR[GP1:91,2] = PR[GP1:90,2] + 31.862;
   1:L PR[91] R[100]mm/sec CNT100;
   1:  PR[GP1:91,1] = PR[GP1:90,1] + -50.094;
   1:  PR[GP1:91,2] = PR[GP1:90,2] + 30.946;
   1:L PR[91] R[100]mm/sec CNT100;
   1:  PR[GP1:91,1] = PR[GP1:90,1] + -54.892;
   1:  PR[GP1:91,2] = PR[GP1:90,2] + 27.974;
   1:L PR[91] R[100]mm/sec CNT100;
   1:  PR[GP1:91,1] = PR[GP1:90,1] + -58.014;
   1:  PR[GP1:91,2] = PR[GP1:90,2] + 25.176;
   1:L PR[91] R[100]mm/sec CNT100;
   1:  PR[GP1:91,1] = PR[GP1:90,1] + -60.994;
   1:  PR[GP1:91,2] = PR[GP1:90,2] + 22.043;
   1:L PR[91] R[100]mm/sec CNT100;
   1:  PR[GP1:91,1] = PR[GP1:90,1] + -63.223;
   1:  PR[GP1:91,2] = PR[GP1:90,2] + 19.149;
   1:L PR[91] R[100]mm/sec CNT100;
   1:  PR[GP1:91,1] = PR[GP1:90,1] + -67.187;
   1:  PR[GP1:91,2] = PR[GP1:90,2] + 11.249;
   1:L PR[91] R[100]mm/sec CNT100;
   1:  PR[GP1:91,1] = PR[GP1:90,1] + -67.953;
   1:  PR[GP1:91,2] = PR[GP1:90,2] + 8.647;
   1:L PR[91] R[100]mm/sec CNT100;
   1:  PR[GP1:91,1] = PR[GP1:90,1] + -68.926;
   1:  PR[GP1:91,2] = PR[GP1:90,2] + 2.403;
   1:L PR[91] R[100]mm/sec CNT100;
   1:  PR[GP1:91,1] = PR[GP1:90,1] + -69.147;
   1:  PR[GP1:91,2] = PR[GP1:90,2] + -0.052;
   1:L PR[91] R[100]mm/sec CNT100;
   1:  PR[GP1:91,1] = PR[GP1:90,1] + -68.181;
   1:  PR[GP1:91,2] = PR[GP1:90,2] + -6.168;
   1:L PR[91] R[100]mm/sec CNT100;
   1:  PR[GP1:91,1] = PR[GP1:90,1] + -67.947;
   1:  PR[GP1:91,2] = PR[GP1:90,2] + -8.810;
   1:L PR[91] R[100]mm/sec CNT100;
   1:  PR[GP1:91,1] = PR[GP1:90,1] + -67.187;
   1:  PR[GP1:91,2] = PR[GP1:90,2] + -11.393;
   1:L PR[91] R[100]mm/sec CNT100;
   1:  PR[GP1:91,1] = PR[GP1:90,1] + -63.223;
   1:  PR[GP1:91,2] = PR[GP1:90,2] + -19.293;
   1:L PR[91] R[100]mm/sec CNT100;
   1:  PR[GP1:91,1] = PR[GP1:90,1] + -60.994;
   1:  PR[GP1:91,2] = PR[GP1:90,2] + -22.187;
   1:L PR[91] R[100]mm/sec CNT100;
   1:  PR[GP1:91,1] = PR[GP1:90,1] + -58.014;
   1:  PR[GP1:91,2] = PR[GP1:90,2] + -25.320;
   1:L PR[91] R[100]mm/sec CNT100;
   1:  PR[GP1:91,1] = PR[GP1:90,1] + -54.902;
   1:  PR[GP1:91,2] = PR[GP1:90,2] + -28.109;
   1:L PR[91] R[100]mm/sec CNT100;
   1:  PR[GP1:91,1] = PR[GP1:90,1] + -52.472;
   1:  PR[GP1:91,2] = PR[GP1:90,2] + -29.476;
   1:L PR[91] R[100]mm/sec CNT100;
   1:  PR[GP1:91,1] = PR[GP1:90,1] + -48.471;
   1:  PR[GP1:91,2] = PR[GP1:90,2] + -32.011;
   1:L PR[91] R[100]mm/sec CNT100;
   1:  PR[GP1:91,1] = PR[GP1:90,1] + -42.650;
   1:  PR[GP1:91,2] = PR[GP1:90,2] + -34.302;
   1:L PR[91] R[100]mm/sec CNT100;
   1:  PR[GP1:91,1] = PR[GP1:90,1] + -35.987;
   1:  PR[GP1:91,2] = PR[GP1:90,2] + -35.739;
   1:L PR[91] R[100]mm/sec CNT100;
   1:  PR[GP1:91,1] = PR[GP1:90,1] + -29.950;
   1:  PR[GP1:91,2] = PR[GP1:90,2] + -35.972;
   1:L PR[91] R[100]mm/sec CNT100;
   1:  PR[GP1:91,1] = PR[GP1:90,1] + -28.271;
   1:  PR[GP1:91,2] = PR[GP1:90,2] + -35.977;
   1:L PR[91] R[100]mm/sec CNT100;
   1:  PR[GP1:91,1] = PR[GP1:90,1] + -22.397;
   1:  PR[GP1:91,2] = PR[GP1:90,2] + -35.210;
   1:L PR[91] R[100]mm/sec CNT100;
   1:  PR[GP1:91,1] = PR[GP1:90,1] + -17.377;
   1:  PR[GP1:91,2] = PR[GP1:90,2] + -33.612;
   1:L PR[91] R[100]mm/sec CNT100;
   1:  PR[GP1:91,1] = PR[GP1:90,1] + -14.378;
   1:  PR[GP1:91,2] = PR[GP1:90,2] + -32.570;
   1:L PR[91] R[100]mm/sec CNT100;
   1:  PR[GP1:91,1] = PR[GP1:90,1] + -9.867;
   1:  PR[GP1:91,2] = PR[GP1:90,2] + -30.210;
   1:L PR[91] R[100]mm/sec CNT100;
   1:  PR[GP1:91,1] = PR[GP1:90,1] + -7.690;
   1:  PR[GP1:91,2] = PR[GP1:90,2] + -28.628;
   1:L PR[91] R[100]mm/sec CNT100;
   1:  PR[GP1:91,1] = PR[GP1:90,1] + -5.321;
   1:  PR[GP1:91,2] = PR[GP1:90,2] + -26.773;
   1:L PR[91] R[100]mm/sec CNT100;
   1:  PR[GP1:91,1] = PR[GP1:90,1] + -3.491;
   1:  PR[GP1:91,2] = PR[GP1:90,2] + -24.651;
   1:L PR[91] R[100]mm/sec CNT100;
   1:  PR[GP1:91,1] = PR[GP1:90,1] + -0.966;
   1:  PR[GP1:91,2] = PR[GP1:90,2] + -24.109;
   1:L PR[91] R[100]mm/sec CNT100;
   1:  PR[GP1:91,1] = PR[GP1:90,1] + 0.764;
   1:  PR[GP1:91,2] = PR[GP1:90,2] + -23.192;
   1:L PR[91] R[100]mm/sec CNT100;
   1:  PR[GP1:91,1] = PR[GP1:90,1] + 3.762;
   1:  PR[GP1:91,2] = PR[GP1:90,2] + -24.714;
   1:L PR[91] R[100]mm/sec CNT100;
   1:  PR[GP1:91,1] = PR[GP1:90,1] + 5.554;
   1:  PR[GP1:91,2] = PR[GP1:90,2] + -26.795;
   1:L PR[91] R[100]mm/sec CNT100;
   1:  PR[GP1:91,1] = PR[GP1:90,1] + 7.912;
   1:  PR[GP1:91,2] = PR[GP1:90,2] + -28.640;
   1:L PR[91] R[100]mm/sec CNT100;
   1:  PR[GP1:91,1] = PR[GP1:90,1] + 10.093;
   1:  PR[GP1:91,2] = PR[GP1:90,2] + -30.225;
   1:L PR[91] R[100]mm/sec CNT100;
   1:  PR[GP1:91,1] = PR[GP1:90,1] + 14.570;
   1:  PR[GP1:91,2] = PR[GP1:90,2] + -32.561;
   1:L PR[91] R[100]mm/sec CNT100;
   1:  PR[GP1:91,1] = PR[GP1:90,1] + 20.104;
   1:  PR[GP1:91,2] = PR[GP1:90,2] + -34.339;
   1:L PR[91] R[100]mm/sec CNT100;
   1:  PR[GP1:91,1] = PR[GP1:90,1] + 22.613;
   1:  PR[GP1:91,2] = PR[GP1:90,2] + -35.207;
   1:L PR[91] R[100]mm/sec CNT100;
   1:  PR[GP1:91,1] = PR[GP1:90,1] + 28.461;
   1:  PR[GP1:91,2] = PR[GP1:90,2] + -35.976;
   1:L PR[91] R[100]mm/sec CNT100;
   1:  PR[GP1:91,1] = PR[GP1:90,1] + 35.264;
   1:  PR[GP1:91,2] = PR[GP1:90,2] + -35.747;
   1:L PR[91] R[100]mm/sec CNT100;
   1:  PR[GP1:91,1] = PR[GP1:90,1] + 36.170;
   1:  PR[GP1:91,2] = PR[GP1:90,2] + -35.743;
   1:L PR[91] R[100]mm/sec CNT100;
   1:  PR[GP1:91,1] = PR[GP1:90,1] + 42.812;
   1:  PR[GP1:91,2] = PR[GP1:90,2] + -34.314;
   1:L PR[91] R[100]mm/sec CNT100;
   1:  PR[GP1:91,1] = PR[GP1:90,1] + 48.671;
   1:  PR[GP1:91,2] = PR[GP1:90,2] + -32.020;
   1:L PR[91] R[100]mm/sec CNT100;
   1:  PR[GP1:91,1] = PR[GP1:90,1] + 50.273;
   1:  PR[GP1:91,2] = PR[GP1:90,2] + -31.110;
   1:L PR[91] R[100]mm/sec CNT100;
   1:  PR[GP1:91,1] = PR[GP1:90,1] + 55.060;
   1:  PR[GP1:91,2] = PR[GP1:90,2] + -28.159;
   1:L PR[91] R[100]mm/sec CNT100;
   1:  PR[GP1:91,1] = PR[GP1:90,1] + 58.179;
   1:  PR[GP1:91,2] = PR[GP1:90,2] + -25.371;
   1:L PR[91] R[100]mm/sec CNT100;
   1:  PR[GP1:91,1] = PR[GP1:90,1] + 61.154;
   1:  PR[GP1:91,2] = PR[GP1:90,2] + -22.233;
   1:L PR[91] R[100]mm/sec CNT100;
   1:  PR[GP1:91,1] = PR[GP1:90,1] + 63.417;
   1:  PR[GP1:91,2] = PR[GP1:90,2] + -19.305;
   1:L PR[91] R[100]mm/sec CNT100;
   1:  PR[GP1:91,1] = PR[GP1:90,1] + 65.893;
   1:  PR[GP1:91,2] = PR[GP1:90,2] + -14.376;
   1:L PR[91] R[100]mm/sec CNT100;
   1:  PR[GP1:91,1] = PR[GP1:90,1] + 67.388;
   1:  PR[GP1:91,2] = PR[GP1:90,2] + -11.446;
   1:L PR[91] R[100]mm/sec CNT100;
   1:  PR[GP1:91,1] = PR[GP1:90,1] + 68.154;
   1:  PR[GP1:91,2] = PR[GP1:90,2] + -8.881;
   1:L PR[91] R[100]mm/sec CNT100;
   1:  PR[GP1:91,1] = PR[GP1:90,1] + 69.128;
   1:  PR[GP1:91,2] = PR[GP1:90,2] + -2.619;
   1:L PR[91] R[100]mm/sec CNT100;
   1:  PR[GP1:91,1] = PR[GP1:90,1] + 69.360;
   1:  PR[GP1:91,2] = PR[GP1:90,2] + -0.092;
   1:L PR[91] R[100]mm/sec CNT100;
   1:  PR[GP1:91,1] = PR[GP1:90,1] + 68.394;
   1:  PR[GP1:91,2] = PR[GP1:90,2] + 6.040;
   1:L PR[91] R[100]mm/sec CNT100;
   1:  PR[GP1:91,1] = PR[GP1:90,1] + 68.148;
   1:  PR[GP1:91,2] = PR[GP1:90,2] + 8.755;
   1:L PR[91] R[100]mm/sec CNT100;
   1:  PR[GP1:91,1] = PR[GP1:90,1] + 67.388;
   1:  PR[GP1:91,2] = PR[GP1:90,2] + 11.304;
   1:L PR[91] R[100]mm/sec CNT100;
   1:  PR[GP1:91,1] = PR[GP1:90,1] + 64.883;
   1:  PR[GP1:91,2] = PR[GP1:90,2] + 16.293;
   1:L PR[91] R[100]mm/sec CNT100;
   1:  PR[GP1:91,1] = PR[GP1:90,1] + 63.418;
   1:  PR[GP1:91,2] = PR[GP1:90,2] + 19.160;
   1:L PR[91] R[100]mm/sec CNT100;
   1:  PR[GP1:91,1] = PR[GP1:90,1] + 61.154;
   1:  PR[GP1:91,2] = PR[GP1:90,2] + 22.089;
   1:L PR[91] R[100]mm/sec CNT100;
   1:  PR[GP1:91,1] = PR[GP1:90,1] + 58.179;
   1:  PR[GP1:91,2] = PR[GP1:90,2] + 25.227;
   1:L PR[91] R[100]mm/sec CNT100;
   1:  PR[GP1:91,1] = PR[GP1:90,1] + 55.069;
   1:  PR[GP1:91,2] = PR[GP1:90,2] + 28.007;
   1:L PR[91] R[100]mm/sec CNT100;
   1:  PR[GP1:91,1] = PR[GP1:90,1] + 52.646;
   1:  PR[GP1:91,2] = PR[GP1:90,2] + 29.368;
   1:L PR[91] R[100]mm/sec CNT100;
   1:  PR[GP1:91,1] = PR[GP1:90,1] + 48.658;
   1:  PR[GP1:91,2] = PR[GP1:90,2] + 31.881;
   1:L PR[91] R[100]mm/sec CNT100;
   1:  PR[GP1:91,1] = PR[GP1:90,1] + 42.812;
   1:  PR[GP1:91,2] = PR[GP1:90,2] + 34.170;
   1:L PR[91] R[100]mm/sec CNT100;
   1:  PR[GP1:91,1] = PR[GP1:90,1] + 36.161;
   1:  PR[GP1:91,2] = PR[GP1:90,2] + 35.601;
   1:L PR[91] R[100]mm/sec CNT100;
   1:  PR[GP1:91,1] = PR[GP1:90,1] + 30.154;
   1:  PR[GP1:91,2] = PR[GP1:90,2] + 35.828;
   1:L PR[91] R[100]mm/sec CNT100;
   1:  PR[GP1:91,1] = PR[GP1:90,1] + 28.473;
   1:  PR[GP1:91,2] = PR[GP1:90,2] + 35.834;
   1:L PR[91] R[100]mm/sec CNT100;
   1:  PR[GP1:91,1] = PR[GP1:90,1] + 22.609;
   1:  PR[GP1:91,2] = PR[GP1:90,2] + 35.063;
   1:L PR[91] R[100]mm/sec CNT100;
   1:  PR[GP1:91,1] = PR[GP1:90,1] + 17.584;
   1:  PR[GP1:91,2] = PR[GP1:90,2] + 33.464;
   1:L PR[91] R[100]mm/sec CNT100;
   1:  PR[GP1:91,1] = PR[GP1:90,1] + 14.581;
   1:  PR[GP1:91,2] = PR[GP1:90,2] + 32.423;
   1:L PR[91] R[100]mm/sec CNT100;
   1:  PR[GP1:91,1] = PR[GP1:90,1] + 10.093;
   1:  PR[GP1:91,2] = PR[GP1:90,2] + 30.081;
   1:L PR[91] R[100]mm/sec CNT100;
   1:  PR[GP1:91,1] = PR[GP1:90,1] + 8.517;
   1:  PR[GP1:91,2] = PR[GP1:90,2] + 28.967;
   1:L PR[91] R[100]mm/sec CNT100;
   1:  PR[GP1:91,1] = PR[GP1:90,1] + 5.831;
   1:  PR[GP1:91,2] = PR[GP1:90,2] + 26.866;
   1:L PR[91] R[100]mm/sec CNT100;
   1:  PR[GP1:91,1] = PR[GP1:90,1] + 3.745;
   1:  PR[GP1:91,2] = PR[GP1:90,2] + 24.438;
   1:L PR[91] R[100]mm/sec CNT100;
   1:  PR[GP1:91,1] = PR[GP1:90,1] + 2.602;
   1:  PR[GP1:91,2] = PR[GP1:90,2] + 23.986;
   1:L PR[91] R[100]mm/sec CNT100;
   1:  PR[GP1:91,1] = PR[GP1:90,1] + 0.877;
   1:  PR[GP1:91,2] = PR[GP1:90,2] + 23.105;
   1:L PR[91] R[100]mm/sec CNT100;
   1:  ! -- Layer/Ebene 79 -- !;
   1:  PR[91] = PR[90];
   1:  PR[GP1:91,1] = PR[GP1:90,1] + -1.566;
   1:  PR[GP1:91,2] = PR[GP1:90,2] + 23.754;
   1:  PR[GP1:91,3] = PR[GP1:90,3] + 48.495;
   1:L PR[91] R[100]mm/sec CNT100;
   1:  PR[GP1:91,1] = PR[GP1:90,1] + -3.518;
   1:  PR[GP1:91,2] = PR[GP1:90,2] + 24.747;
   1:L PR[91] R[100]mm/sec CNT100;
   1:  PR[GP1:91,1] = PR[GP1:90,1] + -5.440;
   1:  PR[GP1:91,2] = PR[GP1:90,2] + 26.981;
   1:L PR[91] R[100]mm/sec CNT100;
   1:  PR[GP1:91,1] = PR[GP1:90,1] + -7.965;
   1:  PR[GP1:91,2] = PR[GP1:90,2] + 28.958;
   1:L PR[91] R[100]mm/sec CNT100;
   1:  PR[GP1:91,1] = PR[GP1:90,1] + -9.656;
   1:  PR[GP1:91,2] = PR[GP1:90,2] + 30.154;
   1:L PR[91] R[100]mm/sec CNT100;
   1:  PR[GP1:91,1] = PR[GP1:90,1] + -14.034;
   1:  PR[GP1:91,2] = PR[GP1:90,2] + 32.444;
   1:L PR[91] R[100]mm/sec CNT100;
   1:  PR[GP1:91,1] = PR[GP1:90,1] + -19.403;
   1:  PR[GP1:91,2] = PR[GP1:90,2] + 34.169;
   1:L PR[91] R[100]mm/sec CNT100;
   1:  PR[GP1:91,1] = PR[GP1:90,1] + -22.210;
   1:  PR[GP1:91,2] = PR[GP1:90,2] + 35.140;
   1:L PR[91] R[100]mm/sec CNT100;
   1:  PR[GP1:91,1] = PR[GP1:90,1] + -27.913;
   1:  PR[GP1:91,2] = PR[GP1:90,2] + 35.885;
   1:L PR[91] R[100]mm/sec CNT100;
   1:  PR[GP1:91,1] = PR[GP1:90,1] + -34.570;
   1:  PR[GP1:91,2] = PR[GP1:90,2] + 35.656;
   1:L PR[91] R[100]mm/sec CNT100;
   1:  PR[GP1:91,1] = PR[GP1:90,1] + -35.811;
   1:  PR[GP1:91,2] = PR[GP1:90,2] + 35.650;
   1:L PR[91] R[100]mm/sec CNT100;
   1:  PR[GP1:91,1] = PR[GP1:90,1] + -42.304;
   1:  PR[GP1:91,2] = PR[GP1:90,2] + 34.249;
   1:L PR[91] R[100]mm/sec CNT100;
   1:  PR[GP1:91,1] = PR[GP1:90,1] + -48.489;
   1:  PR[GP1:91,2] = PR[GP1:90,2] + 31.809;
   1:L PR[91] R[100]mm/sec CNT100;
   1:  PR[GP1:91,1] = PR[GP1:90,1] + -49.470;
   1:  PR[GP1:91,2] = PR[GP1:90,2] + 31.251;
   1:L PR[91] R[100]mm/sec CNT100;
   1:  PR[GP1:91,1] = PR[GP1:90,1] + -54.679;
   1:  PR[GP1:91,2] = PR[GP1:90,2] + 28.024;
   1:L PR[91] R[100]mm/sec CNT100;
   1:  PR[GP1:91,1] = PR[GP1:90,1] + -58.069;
   1:  PR[GP1:91,2] = PR[GP1:90,2] + 24.985;
   1:L PR[91] R[100]mm/sec CNT100;
   1:  PR[GP1:91,1] = PR[GP1:90,1] + -60.627;
   1:  PR[GP1:91,2] = PR[GP1:90,2] + 22.296;
   1:L PR[91] R[100]mm/sec CNT100;
   1:  PR[GP1:91,1] = PR[GP1:90,1] + -63.098;
   1:  PR[GP1:91,2] = PR[GP1:90,2] + 19.088;
   1:L PR[91] R[100]mm/sec CNT100;
   1:  PR[GP1:91,1] = PR[GP1:90,1] + -66.970;
   1:  PR[GP1:91,2] = PR[GP1:90,2] + 11.375;
   1:L PR[91] R[100]mm/sec CNT100;
   1:  PR[GP1:91,1] = PR[GP1:90,1] + -67.836;
   1:  PR[GP1:91,2] = PR[GP1:90,2] + 8.432;
   1:L PR[91] R[100]mm/sec CNT100;
   1:  PR[GP1:91,1] = PR[GP1:90,1] + -68.719;
   1:  PR[GP1:91,2] = PR[GP1:90,2] + 2.766;
   1:L PR[91] R[100]mm/sec CNT100;
   1:  PR[GP1:91,1] = PR[GP1:90,1] + -68.973;
   1:  PR[GP1:91,2] = PR[GP1:90,2] + -0.052;
   1:L PR[91] R[100]mm/sec CNT100;
   1:  PR[GP1:91,1] = PR[GP1:90,1] + -68.094;
   1:  PR[GP1:91,2] = PR[GP1:90,2] + -5.615;
   1:L PR[91] R[100]mm/sec CNT100;
   1:  PR[GP1:91,1] = PR[GP1:90,1] + -67.830;
   1:  PR[GP1:91,2] = PR[GP1:90,2] + -8.596;
   1:L PR[91] R[100]mm/sec CNT100;
   1:  PR[GP1:91,1] = PR[GP1:90,1] + -66.970;
   1:  PR[GP1:91,2] = PR[GP1:90,2] + -11.519;
   1:L PR[91] R[100]mm/sec CNT100;
   1:  PR[GP1:91,1] = PR[GP1:90,1] + -63.098;
   1:  PR[GP1:91,2] = PR[GP1:90,2] + -19.232;
   1:L PR[91] R[100]mm/sec CNT100;
   1:  PR[GP1:91,1] = PR[GP1:90,1] + -60.627;
   1:  PR[GP1:91,2] = PR[GP1:90,2] + -22.440;
   1:L PR[91] R[100]mm/sec CNT100;
   1:  PR[GP1:91,1] = PR[GP1:90,1] + -58.069;
   1:  PR[GP1:91,2] = PR[GP1:90,2] + -25.129;
   1:L PR[91] R[100]mm/sec CNT100;
   1:  PR[GP1:91,1] = PR[GP1:90,1] + -54.689;
   1:  PR[GP1:91,2] = PR[GP1:90,2] + -28.159;
   1:L PR[91] R[100]mm/sec CNT100;
   1:  PR[GP1:91,1] = PR[GP1:90,1] + -52.748;
   1:  PR[GP1:91,2] = PR[GP1:90,2] + -29.251;
   1:L PR[91] R[100]mm/sec CNT100;
   1:  PR[GP1:91,1] = PR[GP1:90,1] + -48.476;
   1:  PR[GP1:91,2] = PR[GP1:90,2] + -31.958;
   1:L PR[91] R[100]mm/sec CNT100;
   1:  PR[GP1:91,1] = PR[GP1:90,1] + -44.874;
   1:  PR[GP1:91,2] = PR[GP1:90,2] + -33.375;
   1:L PR[91] R[100]mm/sec CNT100;
   1:  PR[GP1:91,1] = PR[GP1:90,1] + -42.571;
   1:  PR[GP1:91,2] = PR[GP1:90,2] + -34.300;
   1:L PR[91] R[100]mm/sec CNT100;
   1:  PR[GP1:91,1] = PR[GP1:90,1] + -42.314;
   1:  PR[GP1:91,2] = PR[GP1:90,2] + -34.391;
   1:L PR[91] R[100]mm/sec CNT100;
   1:  PR[GP1:91,1] = PR[GP1:90,1] + -35.799;
   1:  PR[GP1:91,2] = PR[GP1:90,2] + -35.796;
   1:L PR[91] R[100]mm/sec CNT100;
   1:  PR[GP1:91,1] = PR[GP1:90,1] + -29.905;
   1:  PR[GP1:91,2] = PR[GP1:90,2] + -36.023;
   1:L PR[91] R[100]mm/sec CNT100;
   1:  PR[GP1:91,1] = PR[GP1:90,1] + -27.918;
   1:  PR[GP1:91,2] = PR[GP1:90,2] + -36.030;
   1:L PR[91] R[100]mm/sec CNT100;
   1:  PR[GP1:91,1] = PR[GP1:90,1] + -22.198;
   1:  PR[GP1:91,2] = PR[GP1:90,2] + -35.282;
   1:L PR[91] R[100]mm/sec CNT100;
   1:  PR[GP1:91,1] = PR[GP1:90,1] + -17.309;
   1:  PR[GP1:91,2] = PR[GP1:90,2] + -33.726;
   1:L PR[91] R[100]mm/sec CNT100;
   1:  PR[GP1:91,1] = PR[GP1:90,1] + -14.035;
   1:  PR[GP1:91,2] = PR[GP1:90,2] + -32.588;
   1:L PR[91] R[100]mm/sec CNT100;
   1:  PR[GP1:91,1] = PR[GP1:90,1] + -9.656;
   1:  PR[GP1:91,2] = PR[GP1:90,2] + -30.297;
   1:L PR[91] R[100]mm/sec CNT100;
   1:  PR[GP1:91,1] = PR[GP1:90,1] + -7.315;
   1:  PR[GP1:91,2] = PR[GP1:90,2] + -28.597;
   1:L PR[91] R[100]mm/sec CNT100;
   1:  PR[GP1:91,1] = PR[GP1:90,1] + -5.147;
   1:  PR[GP1:91,2] = PR[GP1:90,2] + -26.899;
   1:L PR[91] R[100]mm/sec CNT100;
   1:  PR[GP1:91,1] = PR[GP1:90,1] + -3.462;
   1:  PR[GP1:91,2] = PR[GP1:90,2] + -24.944;
   1:L PR[91] R[100]mm/sec CNT100;
   1:  PR[GP1:91,1] = PR[GP1:90,1] + -0.800;
   1:  PR[GP1:91,2] = PR[GP1:90,2] + -24.372;
   1:L PR[91] R[100]mm/sec CNT100;
   1:  PR[GP1:91,1] = PR[GP1:90,1] + 0.805;
   1:  PR[GP1:91,2] = PR[GP1:90,2] + -23.522;
   1:L PR[91] R[100]mm/sec CNT100;
   1:  PR[GP1:91,1] = PR[GP1:90,1] + 3.732;
   1:  PR[GP1:91,2] = PR[GP1:90,2] + -25.007;
   1:L PR[91] R[100]mm/sec CNT100;
   1:  PR[GP1:91,1] = PR[GP1:90,1] + 5.379;
   1:  PR[GP1:91,2] = PR[GP1:90,2] + -26.919;
   1:L PR[91] R[100]mm/sec CNT100;
   1:  PR[GP1:91,1] = PR[GP1:90,1] + 7.537;
   1:  PR[GP1:91,2] = PR[GP1:90,2] + -28.608;
   1:L PR[91] R[100]mm/sec CNT100;
   1:  PR[GP1:91,1] = PR[GP1:90,1] + 9.882;
   1:  PR[GP1:91,2] = PR[GP1:90,2] + -30.311;
   1:L PR[91] R[100]mm/sec CNT100;
   1:  PR[GP1:91,1] = PR[GP1:90,1] + 14.228;
   1:  PR[GP1:91,2] = PR[GP1:90,2] + -32.579;
   1:L PR[91] R[100]mm/sec CNT100;
   1:  PR[GP1:91,1] = PR[GP1:90,1] + 19.602;
   1:  PR[GP1:91,2] = PR[GP1:90,2] + -34.306;
   1:L PR[91] R[100]mm/sec CNT100;
   1:  PR[GP1:91,1] = PR[GP1:90,1] + 22.414;
   1:  PR[GP1:91,2] = PR[GP1:90,2] + -35.280;
   1:L PR[91] R[100]mm/sec CNT100;
   1:  PR[GP1:91,1] = PR[GP1:90,1] + 28.109;
   1:  PR[GP1:91,2] = PR[GP1:90,2] + -36.028;
   1:L PR[91] R[100]mm/sec CNT100;
   1:  PR[GP1:91,1] = PR[GP1:90,1] + 34.736;
   1:  PR[GP1:91,2] = PR[GP1:90,2] + -35.805;
   1:L PR[91] R[100]mm/sec CNT100;
   1:  PR[GP1:91,1] = PR[GP1:90,1] + 35.982;
   1:  PR[GP1:91,2] = PR[GP1:90,2] + -35.800;
   1:L PR[91] R[100]mm/sec CNT100;
   1:  PR[GP1:91,1] = PR[GP1:90,1] + 42.467;
   1:  PR[GP1:91,2] = PR[GP1:90,2] + -34.404;
   1:L PR[91] R[100]mm/sec CNT100;
   1:  PR[GP1:91,1] = PR[GP1:90,1] + 48.673;
   1:  PR[GP1:91,2] = PR[GP1:90,2] + -31.968;
   1:L PR[91] R[100]mm/sec CNT100;
   1:  PR[GP1:91,1] = PR[GP1:90,1] + 49.646;
   1:  PR[GP1:91,2] = PR[GP1:90,2] + -31.415;
   1:L PR[91] R[100]mm/sec CNT100;
   1:  PR[GP1:91,1] = PR[GP1:90,1] + 54.843;
   1:  PR[GP1:91,2] = PR[GP1:90,2] + -28.212;
   1:L PR[91] R[100]mm/sec CNT100;
   1:  PR[GP1:91,1] = PR[GP1:90,1] + 58.230;
   1:  PR[GP1:91,2] = PR[GP1:90,2] + -25.184;
   1:L PR[91] R[100]mm/sec CNT100;
   1:  PR[GP1:91,1] = PR[GP1:90,1] + 60.782;
   1:  PR[GP1:91,2] = PR[GP1:90,2] + -22.493;
   1:L PR[91] R[100]mm/sec CNT100;
   1:  PR[GP1:91,1] = PR[GP1:90,1] + 63.290;
   1:  PR[GP1:91,2] = PR[GP1:90,2] + -19.247;
   1:L PR[91] R[100]mm/sec CNT100;
   1:  PR[GP1:91,1] = PR[GP1:90,1] + 65.483;
   1:  PR[GP1:91,2] = PR[GP1:90,2] + -14.883;
   1:L PR[91] R[100]mm/sec CNT100;
   1:  PR[GP1:91,1] = PR[GP1:90,1] + 67.170;
   1:  PR[GP1:91,2] = PR[GP1:90,2] + -11.576;
   1:L PR[91] R[100]mm/sec CNT100;
   1:  PR[GP1:91,1] = PR[GP1:90,1] + 68.036;
   1:  PR[GP1:91,2] = PR[GP1:90,2] + -8.675;
   1:L PR[91] R[100]mm/sec CNT100;
   1:  PR[GP1:91,1] = PR[GP1:90,1] + 68.920;
   1:  PR[GP1:91,2] = PR[GP1:90,2] + -2.992;
   1:L PR[91] R[100]mm/sec CNT100;
   1:  PR[GP1:91,1] = PR[GP1:90,1] + 69.186;
   1:  PR[GP1:91,2] = PR[GP1:90,2] + -0.092;
   1:L PR[91] R[100]mm/sec CNT100;
   1:  PR[GP1:91,1] = PR[GP1:90,1] + 68.307;
   1:  PR[GP1:91,2] = PR[GP1:90,2] + 5.486;
   1:L PR[91] R[100]mm/sec CNT100;
   1:  PR[GP1:91,1] = PR[GP1:90,1] + 68.030;
   1:  PR[GP1:91,2] = PR[GP1:90,2] + 8.549;
   1:L PR[91] R[100]mm/sec CNT100;
   1:  PR[GP1:91,1] = PR[GP1:90,1] + 67.169;
   1:  PR[GP1:91,2] = PR[GP1:90,2] + 11.434;
   1:L PR[91] R[100]mm/sec CNT100;
   1:  PR[GP1:91,1] = PR[GP1:90,1] + 64.914;
   1:  PR[GP1:91,2] = PR[GP1:90,2] + 15.926;
   1:L PR[91] R[100]mm/sec CNT100;
   1:  PR[GP1:91,1] = PR[GP1:90,1] + 63.291;
   1:  PR[GP1:91,2] = PR[GP1:90,2] + 19.102;
   1:L PR[91] R[100]mm/sec CNT100;
   1:  PR[GP1:91,1] = PR[GP1:90,1] + 60.782;
   1:  PR[GP1:91,2] = PR[GP1:90,2] + 22.349;
   1:L PR[91] R[100]mm/sec CNT100;
   1:  PR[GP1:91,1] = PR[GP1:90,1] + 58.230;
   1:  PR[GP1:91,2] = PR[GP1:90,2] + 25.040;
   1:L PR[91] R[100]mm/sec CNT100;
   1:  PR[GP1:91,1] = PR[GP1:90,1] + 54.852;
   1:  PR[GP1:91,2] = PR[GP1:90,2] + 28.059;
   1:L PR[91] R[100]mm/sec CNT100;
   1:  PR[GP1:91,1] = PR[GP1:90,1] + 52.919;
   1:  PR[GP1:91,2] = PR[GP1:90,2] + 29.145;
   1:L PR[91] R[100]mm/sec CNT100;
   1:  PR[GP1:91,1] = PR[GP1:90,1] + 48.660;
   1:  PR[GP1:91,2] = PR[GP1:90,2] + 31.829;
   1:L PR[91] R[100]mm/sec CNT100;
   1:  PR[GP1:91,1] = PR[GP1:90,1] + 45.088;
   1:  PR[GP1:91,2] = PR[GP1:90,2] + 33.227;
   1:L PR[91] R[100]mm/sec CNT100;
   1:  PR[GP1:91,1] = PR[GP1:90,1] + 42.740;
   1:  PR[GP1:91,2] = PR[GP1:90,2] + 34.166;
   1:L PR[91] R[100]mm/sec CNT100;
   1:  PR[GP1:91,1] = PR[GP1:90,1] + 42.477;
   1:  PR[GP1:91,2] = PR[GP1:90,2] + 34.258;
   1:L PR[91] R[100]mm/sec CNT100;
   1:  PR[GP1:91,1] = PR[GP1:90,1] + 35.974;
   1:  PR[GP1:91,2] = PR[GP1:90,2] + 35.658;
   1:L PR[91] R[100]mm/sec CNT100;
   1:  PR[GP1:91,1] = PR[GP1:90,1] + 30.108;
   1:  PR[GP1:91,2] = PR[GP1:90,2] + 35.879;
   1:L PR[91] R[100]mm/sec CNT100;
   1:  PR[GP1:91,1] = PR[GP1:90,1] + 28.121;
   1:  PR[GP1:91,2] = PR[GP1:90,2] + 35.886;
   1:L PR[91] R[100]mm/sec CNT100;
   1:  PR[GP1:91,1] = PR[GP1:90,1] + 22.411;
   1:  PR[GP1:91,2] = PR[GP1:90,2] + 35.135;
   1:L PR[91] R[100]mm/sec CNT100;
   1:  PR[GP1:91,1] = PR[GP1:90,1] + 17.516;
   1:  PR[GP1:91,2] = PR[GP1:90,2] + 33.578;
   1:L PR[91] R[100]mm/sec CNT100;
   1:  PR[GP1:91,1] = PR[GP1:90,1] + 14.240;
   1:  PR[GP1:91,2] = PR[GP1:90,2] + 32.442;
   1:L PR[91] R[100]mm/sec CNT100;
   1:  PR[GP1:91,1] = PR[GP1:90,1] + 9.882;
   1:  PR[GP1:91,2] = PR[GP1:90,2] + 30.168;
